LIN {X 0,Y 368.997,Z 325.512,A -85,B 0,C 180,E1 -12767.906,E2 -12767.906} C_VEL
LIN {X 0,Y 369.139,Z 325.499,A -85,B 0,C 180,E1 -12771.892,E2 -12771.892} C_VEL
LIN {X 0,Y 369.12,Z 325.495,A -85,B 0,C 180,E1 -12774.537,E2 -12774.537} C_VEL
LIN {X 0,Y 369.293,Z 325.485,A -85,B 0,C 180,E1 -12777.819,E2 -12777.819} C_VEL
LIN {X 0,Y 369.298,Z 325.479,A -85,B 0,C 180,E1 -12782.181,E2 -12782.181} C_VEL
LIN {X 0,Y 369.147,Z 325.492,A -85,B 0,C 180,E1 -12786.559,E2 -12786.559} C_VEL
LIN {X 0,Y 369.056,Z 325.512,A -85,B 0,C 180,E1 -12789.869,E2 -12789.869} C_VEL
LIN {X 0,Y 369.031,Z 325.503,A -85,B 0,C 180,E1 -12793.772,E2 -12793.772} C_VEL
LIN {X 0,Y 368.985,Z 325.524,A -85,B 0,C 180,E1 -12797.743,E2 -12797.743} C_VEL
LIN {X 0,Y 368.904,Z 325.52,A -85,B 0,C 180,E1 -12801.221,E2 -12801.221} C_VEL
LIN {X 0,Y 368.905,Z 325.533,A -85,B 0,C 180,E1 -12803.875,E2 -12803.875} C_VEL
LIN {X 0,Y 368.852,Z 325.519,A -85,B 0,C 180,E1 -12807.213,E2 -12807.213} C_VEL
LIN {X 0,Y 368.887,Z 325.493,A -85,B 0,C 180,E1 -12809.693,E2 -12809.693} C_VEL
LIN {X 0,Y 368.891,Z 325.526,A -85,B 0,C 180,E1 -12813.043,E2 -12813.043} C_VEL
LIN {X 0,Y 368.911,Z 325.525,A -85,B 0,C 180,E1 -12816.198,E2 -12816.198} C_VEL
LIN {X 0,Y 368.869,Z 325.507,A -85,B 0,C 180,E1 -12818.958,E2 -12818.958} C_VEL
LIN {X 0,Y 368.855,Z 325.537,A -85,B 0,C 180,E1 -12822.006,E2 -12822.006} C_VEL
LIN {X 0,Y 368.87,Z 325.527,A -85,B 0,C 180,E1 -12825.175,E2 -12825.175} C_VEL
LIN {X 0,Y 368.857,Z 325.529,A -85,B 0,C 180,E1 -12828.175,E2 -12828.175} C_VEL
LIN {X 0,Y 368.874,Z 325.529,A -85,B 0,C 180,E1 -12831.367,E2 -12831.367} C_VEL
LIN {X 0,Y 368.929,Z 325.531,A -85,B 0,C 180,E1 -12835.146,E2 -12835.146} C_VEL
LIN {X 0,Y 368.912,Z 325.531,A -85,B 0,C 180,E1 -12839.046,E2 -12839.046} C_VEL
LIN {X 0,Y 368.906,Z 325.505,A -85,B 0,C 180,E1 -12841.558,E2 -12841.558} C_VEL
LIN {X 0,Y 368.922,Z 325.534,A -85,B 0,C 180,E1 -12845.223,E2 -12845.223} C_VEL
LIN {X 0,Y 368.933,Z 325.664,A -85,B 0,C 180,E1 -12848.554,E2 -12848.554} C_VEL
LIN {X 0,Y 369.139,Z 326.592,A -85,B 0,C 180,E1 -12848.752,E2 -12848.752} C_VEL
LIN {X 0,Y 377.458,Z 346.32,A -85,B 0,C 180,E1 -12849.683,E2 -12849.683} C_VEL
LIN {X 0,Y 376.795,Z 405.29,A -85,B 0,C 180,E1 -12850.834,E2 -12850.834} C_VEL
LIN {X 0,Y 376.624,Z 418.447,A -85,B 0,C 180,E1 -12851.267,E2 -12851.267} C_VEL
LIN {X 0,Y 376.25,Z 430.983,A -85,B 0,C 180,E1 -12851.909,E2 -12851.909} C_VEL
LIN {X 0,Y 375.666,Z 442.722,A -85,B 0,C 180,E1 -12852.722,E2 -12852.722} C_VEL
LIN {X 0,Y 374.827,Z 453.399,A -85,B 0,C 180,E1 -12853.666,E2 -12853.666} C_VEL
LIN {X 0,Y 373.891,Z 464.248,A -85,B 0,C 180,E1 -12854.882,E2 -12854.882} C_VEL
LIN {X 0,Y 373.107,Z 473.023,A -85,B 0,C 180,E1 -12856.104,E2 -12856.104} C_VEL
LIN {X 0,Y 372.364,Z 481.054,A -85,B 0,C 180,E1 -12857.464,E2 -12857.464} C_VEL
LIN {X 0,Y 371.492,Z 488.922,A -85,B 0,C 180,E1 -12859.095,E2 -12859.095} C_VEL
LIN {X 0,Y 370.759,Z 494.835,A -85,B 0,C 180,E1 -12860.615,E2 -12860.615} C_VEL
LIN {X 0,Y 370.256,Z 500.214,A -85,B 0,C 180,E1 -12862.365,E2 -12862.365} C_VEL
LIN {X 0,Y 369.648,Z 504.11,A -85,B 0,C 180,E1 -12863.998,E2 -12863.998} C_VEL
LIN {X 0,Y 369.219,Z 506.981,A -85,B 0,C 180,E1 -12865.633,E2 -12865.633} C_VEL
LIN {X 0,Y 369.225,Z 508.328,A -85,B 0,C 180,E1 -12866.727,E2 -12866.727} C_VEL
LIN {X 0,Y 369.048,Z 509.31,A -85,B 0,C 180,E1 -12867.817,E2 -12867.817} C_VEL
LIN {X 0,Y 369.11,Z 509.891,A -85,B 0,C 180,E1 -12868.909,E2 -12868.909} C_VEL
LIN {X 0,Y 369.091,Z 510.119,A -85,B 0,C 180,E1 -12870,E2 -12870} C_VEL
LIN {X 0,Y 369.11,Z 509.934,A -85,B 0,C 180,E1 -12871.091,E2 -12871.091} C_VEL
LIN {X 0,Y 369.047,Z 509.38,A -85,B 0,C 180,E1 -12872.183,E2 -12872.183} C_VEL
LIN {X 0,Y 369.221,Z 508.427,A -85,B 0,C 180,E1 -12873.274,E2 -12873.274} C_VEL
LIN {X 0,Y 369.209,Z 507.125,A -85,B 0,C 180,E1 -12874.367,E2 -12874.367} C_VEL
LIN {X 0,Y 369.643,Z 504.306,A -85,B 0,C 180,E1 -12876.002,E2 -12876.002} C_VEL
LIN {X 0,Y 370.232,Z 500.48,A -85,B 0,C 180,E1 -12877.636,E2 -12877.636} C_VEL
LIN {X 0,Y 370.699,Z 495.402,A -85,B 0,C 180,E1 -12879.328,E2 -12879.328} C_VEL
LIN {X 0,Y 371.612,Z 488.165,A -85,B 0,C 180,E1 -12881.177,E2 -12881.177} C_VEL
LIN {X 0,Y 372.522,Z 480.138,A -85,B 0,C 180,E1 -12882.807,E2 -12882.807} C_VEL
LIN {X 0,Y 373.293,Z 471.916,A -85,B 0,C 180,E1 -12884.167,E2 -12884.167} C_VEL
LIN {X 0,Y 374.07,Z 462.889,A -85,B 0,C 180,E1 -12885.389,E2 -12885.389} C_VEL
LIN {X 0,Y 375.061,Z 452.378,A -85,B 0,C 180,E1 -12886.527,E2 -12886.527} C_VEL
LIN {X 0,Y 375.803,Z 440.712,A -85,B 0,C 180,E1 -12887.537,E2 -12887.537} C_VEL
LIN {X 0,Y 376.419,Z 429.269,A -85,B 0,C 180,E1 -12888.294,E2 -12888.294} C_VEL
LIN {X 0,Y 376.696,Z 416.398,A -85,B 0,C 180,E1 -12888.915,E2 -12888.915} C_VEL
LIN {X 0,Y 376.801,Z 402.594,A -85,B 0,C 180,E1 -12889.333,E2 -12889.333} C_VEL
LIN {X 0,Y 376.774,Z 399.485,A -85,B 0,C 180,E1 -12889.399,E2 -12889.399} C_VEL
LIN {X 0,Y 376.147,Z 393.69,A -85,B 0,C 180,E1 -12889.55,E2 -12889.55} C_VEL
LIN {X 0,Y 371.047,Z 375.043,A -85,B 0,C 180,E1 -12890.224,E2 -12890.224} C_VEL
LIN {X 0,Y 370.502,Z 369.246,A -85,B 0,C 180,E1 -12890.375,E2 -12890.375} C_VEL
LIN {X 0,Y 370.808,Z 347.992,A -85,B 0,C 180,E1 -12890.79,E2 -12890.79} C_VEL
LIN {X 0,Y 362.473,Z 328.467,A -85,B 0,C 180,E1 -12891.729,E2 -12891.729} C_VEL
LIN {X 0,Y 361.96,Z 326.942,A -85,B 0,C 180,E1 -12891.863,E2 -12891.863} C_VEL
LIN {X 0,Y 361.876,Z 326.425,A -85,B 0,C 180,E1 -12892.096,E2 -12892.096} C_VEL
LIN {X 0,Y 361.879,Z 326.4,A -85,B 0,C 180,E1 -12895.293,E2 -12895.293} C_VEL
LIN {X 0,Y 361.855,Z 326.391,A -85,B 0,C 180,E1 -12899.073,E2 -12899.073} C_VEL
LIN {X 0,Y 361.844,Z 326.402,A -85,B 0,C 180,E1 -12902.944,E2 -12902.944} C_VEL
LIN {X 0,Y 361.862,Z 326.408,A -85,B 0,C 180,E1 -12905.637,E2 -12905.637} C_VEL
LIN {X 0,Y 361.823,Z 326.411,A -85,B 0,C 180,E1 -12909.017,E2 -12909.017} C_VEL
LIN {X 0,Y 361.826,Z 326.393,A -85,B 0,C 180,E1 -12912.829,E2 -12912.829} C_VEL
LIN {X 0,Y 361.81,Z 326.414,A -85,B 0,C 180,E1 -12915.947,E2 -12915.947} C_VEL
LIN {X 0,Y 361.806,Z 326.401,A -85,B 0,C 180,E1 -12919.249,E2 -12919.249} C_VEL
LIN {X 0,Y 361.859,Z 326.397,A -85,B 0,C 180,E1 -12922.981,E2 -12922.981} C_VEL
LIN {X 0,Y 361.854,Z 326.406,A -85,B 0,C 180,E1 -12926.63,E2 -12926.63} C_VEL
LIN {X 0,Y 361.842,Z 326.373,A -85,B 0,C 180,E1 -12929.669,E2 -12929.669} C_VEL
LIN {X 0,Y 361.849,Z 326.4,A -85,B 0,C 180,E1 -12933.467,E2 -12933.467} C_VEL
LIN {X 0,Y 361.855,Z 326.406,A -85,B 0,C 180,E1 -12937.142,E2 -12937.142} C_VEL
LIN {X 0,Y 361.869,Z 326.407,A -85,B 0,C 180,E1 -12940.721,E2 -12940.721} C_VEL
LIN {X 0,Y 361.933,Z 326.393,A -85,B 0,C 180,E1 -12944.225,E2 -12944.225} C_VEL
LIN {X 0,Y 361.993,Z 326.384,A -85,B 0,C 180,E1 -12946.527,E2 -12946.527} C_VEL
LIN {X 0,Y 361.99,Z 326.392,A -85,B 0,C 180,E1 -12949.937,E2 -12949.937} C_VEL
LIN {X 0,Y 362.108,Z 326.37,A -85,B 0,C 180,E1 -12953.313,E2 -12953.313} C_VEL
LIN {X 0,Y 362.261,Z 326.355,A -85,B 0,C 180,E1 -12957.776,E2 -12957.776} C_VEL
LIN {X 0,Y 362.256,Z 326.361,A -85,B 0,C 180,E1 -12962.224,E2 -12962.224} C_VEL
LIN {X 0,Y 362.133,Z 326.364,A -85,B 0,C 180,E1 -12966.687,E2 -12966.687} C_VEL
LIN {X 0,Y 361.989,Z 326.395,A -85,B 0,C 180,E1 -12970.063,E2 -12970.063} C_VEL
LIN {X 0,Y 361.992,Z 326.382,A -85,B 0,C 180,E1 -12973.899,E2 -12973.899} C_VEL
LIN {X 0,Y 361.922,Z 326.399,A -85,B 0,C 180,E1 -12976.935,E2 -12976.935} C_VEL
LIN {X 0,Y 361.877,Z 326.381,A -85,B 0,C 180,E1 -12980.461,E2 -12980.461} C_VEL
LIN {X 0,Y 361.855,Z 326.41,A -85,B 0,C 180,E1 -12984.102,E2 -12984.102} C_VEL
LIN {X 0,Y 361.837,Z 326.397,A -85,B 0,C 180,E1 -12987.785,E2 -12987.785} C_VEL
LIN {X 0,Y 361.842,Z 326.411,A -85,B 0,C 180,E1 -12991.286,E2 -12991.286} C_VEL
LIN {X 0,Y 361.846,Z 326.399,A -85,B 0,C 180,E1 -12994.281,E2 -12994.281} C_VEL
LIN {X 0,Y 361.852,Z 326.41,A -85,B 0,C 180,E1 -12997.222,E2 -12997.222} C_VEL
LIN {X 0,Y 361.807,Z 326.416,A -85,B 0,C 180,E1 -13000.751,E2 -13000.751} C_VEL
LIN {X 0,Y 361.806,Z 326.386,A -85,B 0,C 180,E1 -13004.37,E2 -13004.37} C_VEL
LIN {X 0,Y 361.819,Z 326.414,A -85,B 0,C 180,E1 -13007.571,E2 -13007.571} C_VEL
LIN {X 0,Y 361.839,Z 326.402,A -85,B 0,C 180,E1 -13011.572,E2 -13011.572} C_VEL
LIN {X 0,Y 361.91,Z 326.58,A -85,B 0,C 180,E1 -13014.953,E2 -13014.953} C_VEL
LIN {X 0,Y 364.912,Z 338.861,A -85,B 0,C 180,E1 -13017.597,E2 -13017.597} C_VEL
LIN {X 0,Y 367.691,Z 351.772,A -85,B 0,C 180,E1 -13020.201,E2 -13020.201} C_VEL
LIN {X 0,Y 367.318,Z 358.573,A -85,B 0,C 180,E1 -13021.424,E2 -13021.424} C_VEL
LIN {X 0,Y 365.124,Z 381.961,A -85,B 0,C 180,E1 -13025.554,E2 -13025.554} C_VEL
LIN {X 0,Y 364.057,Z 395.066,A -85,B 0,C 180,E1 -13027.831,E2 -13027.831} C_VEL
LIN {X 0,Y 367.984,Z 428.586,A -85,B 0,C 180,E1 -13028.774,E2 -13028.774} C_VEL
LIN {X 0,Y 369.463,Z 445.477,A -85,B 0,C 180,E1 -13029.201,E2 -13029.201} C_VEL
LIN {X 0,Y 368.499,Z 505.753,A -85,B 0,C 180,E1 -13030.395,E2 -13030.395} C_VEL
LIN {X 0,Y 367.813,Z 519.02,A -85,B 0,C 180,E1 -13030.864,E2 -13030.864} C_VEL
LIN {X 0,Y 366.828,Z 532.347,A -85,B 0,C 180,E1 -13031.572,E2 -13031.572} C_VEL
LIN {X 0,Y 365.679,Z 543.548,A -85,B 0,C 180,E1 -13032.38,E2 -13032.38} C_VEL
LIN {X 0,Y 364.475,Z 555.248,A -85,B 0,C 180,E1 -13033.476,E2 -13033.476} C_VEL
LIN {X 0,Y 363.415,Z 564.724,A -85,B 0,C 180,E1 -13034.579,E2 -13034.579} C_VEL
LIN {X 0,Y 362.436,Z 574.494,A -85,B 0,C 180,E1 -13035.973,E2 -13035.973} C_VEL
LIN {X 0,Y 361.919,Z 581.022,A -85,B 0,C 180,E1 -13037.096,E2 -13037.096} C_VEL
LIN {X 0,Y 361.274,Z 589.239,A -85,B 0,C 180,E1 -13038.783,E2 -13038.783} C_VEL
LIN {X 0,Y 360.931,Z 595.87,A -85,B 0,C 180,E1 -13040.473,E2 -13040.473} C_VEL
LIN {X 0,Y 360.895,Z 601.177,A -85,B 0,C 180,E1 -13042.165,E2 -13042.165} C_VEL
LIN {X 0,Y 361.013,Z 605.321,A -85,B 0,C 180,E1 -13043.854,E2 -13043.854} C_VEL
LIN {X 0,Y 361.197,Z 608.397,A -85,B 0,C 180,E1 -13045.536,E2 -13045.536} C_VEL
LIN {X 0,Y 361.295,Z 609.864,A -85,B 0,C 180,E1 -13046.655,E2 -13046.655} C_VEL
LIN {X 0,Y 361.693,Z 611.588,A -85,B 0,C 180,E1 -13048.887,E2 -13048.887} C_VEL
LIN {X 0,Y 361.754,Z 611.819,A -85,B 0,C 180,E1 -13050,E2 -13050} C_VEL
LIN {X 0,Y 361.694,Z 611.584,A -85,B 0,C 180,E1 -13051.113,E2 -13051.113} C_VEL
LIN {X 0,Y 361.299,Z 609.858,A -85,B 0,C 180,E1 -13053.345,E2 -13053.345} C_VEL
LIN {X 0,Y 361.21,Z 608.388,A -85,B 0,C 180,E1 -13054.464,E2 -13054.464} C_VEL
LIN {X 0,Y 361.035,Z 605.305,A -85,B 0,C 180,E1 -13056.146,E2 -13056.146} C_VEL
LIN {X 0,Y 360.904,Z 601.15,A -85,B 0,C 180,E1 -13057.834,E2 -13057.834} C_VEL
LIN {X 0,Y 360.973,Z 594.801,A -85,B 0,C 180,E1 -13059.808,E2 -13059.808} C_VEL
LIN {X 0,Y 361.376,Z 587.926,A -85,B 0,C 180,E1 -13061.498,E2 -13061.498} C_VEL
LIN {X 0,Y 361.914,Z 580.962,A -85,B 0,C 180,E1 -13062.904,E2 -13062.904} C_VEL
LIN {X 0,Y 362.7,Z 571.813,A -85,B 0,C 180,E1 -13064.427,E2 -13064.427} C_VEL
LIN {X 0,Y 363.585,Z 562.451,A -85,B 0,C 180,E1 -13065.701,E2 -13065.701} C_VEL
LIN {X 0,Y 364.898,Z 551.055,A -85,B 0,C 180,E1 -13066.936,E2 -13066.936} C_VEL
LIN {X 0,Y 366.036,Z 539.916,A -85,B 0,C 180,E1 -13067.891,E2 -13067.891} C_VEL
LIN {X 0,Y 367.224,Z 527.607,A -85,B 0,C 180,E1 -13068.697,E2 -13068.697} C_VEL
LIN {X 0,Y 368.076,Z 514.653,A -85,B 0,C 180,E1 -13069.303,E2 -13069.303} C_VEL
LIN {X 0,Y 368.541,Z 500.894,A -85,B 0,C 180,E1 -13069.712,E2 -13069.712} C_VEL
LIN {X 0,Y 369.37,Z 443.517,A -85,B 0,C 180,E1 -13070.83,E2 -13070.83} C_VEL
LIN {X 0,Y 365.882,Z 410.175,A -85,B 0,C 180,E1 -13071.711,E2 -13071.711} C_VEL
LIN {X 0,Y 364.018,Z 394.864,A -85,B 0,C 180,E1 -13072.173,E2 -13072.173} C_VEL
LIN {X 0,Y 365.701,Z 374.774,A -85,B 0,C 180,E1 -13075.703,E2 -13075.703} C_VEL
LIN {X 0,Y 367.61,Z 355.111,A -85,B 0,C 180,E1 -13079.176,E2 -13079.176} C_VEL
LIN {X 0,Y 367.643,Z 351.679,A -85,B 0,C 180,E1 -13079.803,E2 -13079.803} C_VEL
LIN {X 0,Y 364.613,Z 337.52,A -85,B 0,C 180,E1 -13082.663,E2 -13082.663} C_VEL
LIN {X 0,Y 361.91,Z 326.536,A -85,B 0,C 180,E1 -13085.047,E2 -13085.047} C_VEL
LIN {X 0,Y 361.839,Z 326.403,A -85,B 0,C 180,E1 -13088.428,E2 -13088.428} C_VEL
LIN {X 0,Y 361.819,Z 326.415,A -85,B 0,C 180,E1 -13092.429,E2 -13092.429} C_VEL
LIN {X 0,Y 361.808,Z 326.39,A -85,B 0,C 180,E1 -13095.947,E2 -13095.947} C_VEL
LIN {X 0,Y 361.807,Z 326.417,A -85,B 0,C 180,E1 -13099.249,E2 -13099.249} C_VEL
LIN {X 0,Y 361.855,Z 326.355,A -85,B 0,C 180,E1 -13102.98,E2 -13102.98} C_VEL
LIN {X 0,Y 361.853,Z 326.406,A -85,B 0,C 180,E1 -13106.631,E2 -13106.631} C_VEL
LIN {X 0,Y 361.851,Z 326.406,A -85,B 0,C 180,E1 -13109.67,E2 -13109.67} C_VEL
LIN {X 0,Y 361.86,Z 326.403,A -85,B 0,C 180,E1 -13113.468,E2 -13113.468} C_VEL
LIN {X 0,Y 361.87,Z 326.403,A -85,B 0,C 180,E1 -13117.143,E2 -13117.143} C_VEL
LIN {X 0,Y 361.898,Z 326.39,A -85,B 0,C 180,E1 -13120.723,E2 -13120.723} C_VEL
LIN {X 0,Y 361.927,Z 326.399,A -85,B 0,C 180,E1 -13123.066,E2 -13123.066} C_VEL
LIN {X 0,Y 361.993,Z 326.379,A -85,B 0,C 180,E1 -13126.528,E2 -13126.528} C_VEL
LIN {X 0,Y 361.992,Z 326.396,A -85,B 0,C 180,E1 -13129.937,E2 -13129.937} C_VEL
LIN {X 0,Y 362.134,Z 326.365,A -85,B 0,C 180,E1 -13133.313,E2 -13133.313} C_VEL
LIN {X 0,Y 362.256,Z 326.362,A -85,B 0,C 180,E1 -13137.776,E2 -13137.776} C_VEL
LIN {X 0,Y 362.261,Z 326.355,A -85,B 0,C 180,E1 -13142.224,E2 -13142.224} C_VEL
LIN {X 0,Y 362.111,Z 326.369,A -85,B 0,C 180,E1 -13146.687,E2 -13146.687} C_VEL
LIN {X 0,Y 361.993,Z 326.392,A -85,B 0,C 180,E1 -13150.063,E2 -13150.063} C_VEL
LIN {X 0,Y 361.992,Z 326.379,A -85,B 0,C 180,E1 -13153.899,E2 -13153.899} C_VEL
LIN {X 0,Y 361.921,Z 326.398,A -85,B 0,C 180,E1 -13156.935,E2 -13156.935} C_VEL
LIN {X 0,Y 361.877,Z 326.395,A -85,B 0,C 180,E1 -13160.462,E2 -13160.462} C_VEL
LIN {X 0,Y 361.856,Z 326.409,A -85,B 0,C 180,E1 -13164.102,E2 -13164.102} C_VEL
LIN {X 0,Y 361.829,Z 326.385,A -85,B 0,C 180,E1 -13167.786,E2 -13167.786} C_VEL
LIN {X 0,Y 361.84,Z 326.383,A -85,B 0,C 180,E1 -13171.285,E2 -13171.285} C_VEL
LIN {X 0,Y 361.849,Z 326.41,A -85,B 0,C 180,E1 -13174.281,E2 -13174.281} C_VEL
LIN {X 0,Y 361.855,Z 326.396,A -85,B 0,C 180,E1 -13177.222,E2 -13177.222} C_VEL
LIN {X 0,Y 361.806,Z 326.399,A -85,B 0,C 180,E1 -13180.751,E2 -13180.751} C_VEL
LIN {X 0,Y 361.809,Z 326.413,A -85,B 0,C 180,E1 -13184.37,E2 -13184.37} C_VEL
LIN {X 0,Y 361.819,Z 326.396,A -85,B 0,C 180,E1 -13187.571,E2 -13187.571} C_VEL
LIN {X 0,Y 361.84,Z 326.402,A -85,B 0,C 180,E1 -13191.573,E2 -13191.573} C_VEL
LIN {X 0,Y 361.868,Z 326.407,A -85,B 0,C 180,E1 -13194.657,E2 -13194.657} C_VEL
LIN {X 0,Y 361.836,Z 326.409,A -85,B 0,C 180,E1 -13198.371,E2 -13198.371} C_VEL
LIN {X 0,Y 361.848,Z 326.394,A -85,B 0,C 180,E1 -13200.951,E2 -13200.951} C_VEL
LIN {X 0,Y 361.879,Z 326.4,A -85,B 0,C 180,E1 -13204.707,E2 -13204.707} C_VEL
LIN {X 0,Y 361.903,Z 326.554,A -85,B 0,C 180,E1 -13208.124,E2 -13208.124} C_VEL
LIN {X 0,Y 362.125,Z 327.56,A -85,B 0,C 180,E1 -13208.321,E2 -13208.321} C_VEL
LIN {X 0,Y 369.789,Z 345.481,A -85,B 0,C 180,E1 -13209.201,E2 -13209.201} C_VEL
LIN {X 0,Y 370.86,Z 348.15,A -85,B 0,C 180,E1 -13209.322,E2 -13209.322} C_VEL
LIN {X 0,Y 370.152,Z 405.371,A -85,B 0,C 180,E1 -13210.454,E2 -13210.454} C_VEL
LIN {X 0,Y 369.988,Z 418.734,A -85,B 0,C 180,E1 -13210.889,E2 -13210.889} C_VEL
LIN {X 0,Y 369.616,Z 430.853,A -85,B 0,C 180,E1 -13211.501,E2 -13211.501} C_VEL
LIN {X 0,Y 368.981,Z 443.151,A -85,B 0,C 180,E1 -13212.354,E2 -13212.354} C_VEL
LIN {X 0,Y 368.203,Z 453.321,A -85,B 0,C 180,E1 -13213.256,E2 -13213.256} C_VEL
LIN {X 0,Y 367.184,Z 464.17,A -85,B 0,C 180,E1 -13214.457,E2 -13214.457} C_VEL
LIN {X 0,Y 366.288,Z 474.004,A -85,B 0,C 180,E1 -13215.84,E2 -13215.84} C_VEL
LIN {X 0,Y 365.506,Z 482.035,A -85,B 0,C 180,E1 -13217.225,E2 -13217.225} C_VEL
LIN {X 0,Y 364.594,Z 489.902,A -85,B 0,C 180,E1 -13218.886,E2 -13218.886} C_VEL
LIN {X 0,Y 363.827,Z 495.815,A -85,B 0,C 180,E1 -13220.435,E2 -13220.435} C_VEL
LIN {X 0,Y 363.292,Z 501.193,A -85,B 0,C 180,E1 -13222.217,E2 -13222.217} C_VEL
LIN {X 0,Y 362.659,Z 505.088,A -85,B 0,C 180,E1 -13223.882,E2 -13223.882} C_VEL
LIN {X 0,Y 362.208,Z 507.96,A -85,B 0,C 180,E1 -13225.549,E2 -13225.549} C_VEL
LIN {X 0,Y 362.207,Z 509.307,A -85,B 0,C 180,E1 -13226.663,E2 -13226.663} C_VEL
LIN {X 0,Y 362.026,Z 510.288,A -85,B 0,C 180,E1 -13227.775,E2 -13227.775} C_VEL
LIN {X 0,Y 362.085,Z 510.869,A -85,B 0,C 180,E1 -13228.888,E2 -13228.888} C_VEL
LIN {X 0,Y 362.065,Z 511.097,A -85,B 0,C 180,E1 -13230,E2 -13230} C_VEL
LIN {X 0,Y 362.085,Z 510.911,A -85,B 0,C 180,E1 -13231.112,E2 -13231.112} C_VEL
LIN {X 0,Y 362.025,Z 510.358,A -85,B 0,C 180,E1 -13232.225,E2 -13232.225} C_VEL
LIN {X 0,Y 362.204,Z 509.404,A -85,B 0,C 180,E1 -13233.337,E2 -13233.337} C_VEL
LIN {X 0,Y 362.198,Z 508.103,A -85,B 0,C 180,E1 -13234.451,E2 -13234.451} C_VEL
LIN {X 0,Y 362.654,Z 505.283,A -85,B 0,C 180,E1 -13236.118,E2 -13236.118} C_VEL
LIN {X 0,Y 363.268,Z 501.457,A -85,B 0,C 180,E1 -13237.783,E2 -13237.783} C_VEL
LIN {X 0,Y 363.765,Z 496.379,A -85,B 0,C 180,E1 -13239.508,E2 -13239.508} C_VEL
LIN {X 0,Y 364.723,Z 489.141,A -85,B 0,C 180,E1 -13241.391,E2 -13241.391} C_VEL
LIN {X 0,Y 365.671,Z 481.113,A -85,B 0,C 180,E1 -13243.051,E2 -13243.051} C_VEL
LIN {X 0,Y 366.481,Z 472.892,A -85,B 0,C 180,E1 -13244.436,E2 -13244.436} C_VEL
LIN {X 0,Y 367.311,Z 463.861,A -85,B 0,C 180,E1 -13245.68,E2 -13245.68} C_VEL
LIN {X 0,Y 368.325,Z 453.353,A -85,B 0,C 180,E1 -13246.838,E2 -13246.838} C_VEL
LIN {X 0,Y 369.087,Z 441.84,A -85,B 0,C 180,E1 -13247.854,E2 -13247.854} C_VEL
LIN {X 0,Y 369.732,Z 430.576,A -85,B 0,C 180,E1 -13248.616,E2 -13248.616} C_VEL
LIN {X 0,Y 370.095,Z 418.263,A -85,B 0,C 180,E1 -13249.229,E2 -13249.229} C_VEL
LIN {X 0,Y 370.183,Z 408.012,A -85,B 0,C 180,E1 -13249.585,E2 -13249.585} C_VEL
LIN {X 0,Y 370.502,Z 369.246,A -85,B 0,C 180,E1 -13250.375,E2 -13250.375} C_VEL
LIN {X 0,Y 370.017,Z 365.384,A -85,B 0,C 180,E1 -13250.483,E2 -13250.483} C_VEL
LIN {X 0,Y 367.762,Z 359.348,A -85,B 0,C 180,E1 -13250.745,E2 -13250.745} C_VEL
LIN {X 0,Y 364.755,Z 352.129,A -85,B 0,C 180,E1 -13251.083,E2 -13251.083} C_VEL
LIN {X 0,Y 364.157,Z 349.57,A -85,B 0,C 180,E1 -13251.175,E2 -13251.175} C_VEL
LIN {X 0,Y 355.034,Z 328.299,A -85,B 0,C 180,E1 -13252.254,E2 -13252.254} C_VEL
LIN {X 0,Y 354.823,Z 327.338,A -85,B 0,C 180,E1 -13252.487,E2 -13252.487} C_VEL
LIN {X 0,Y 354.808,Z 327.266,A -85,B 0,C 180,E1 -13255.834,E2 -13255.834} C_VEL
LIN {X 0,Y 354.792,Z 327.283,A -85,B 0,C 180,E1 -13259.684,E2 -13259.684} C_VEL
LIN {X 0,Y 354.783,Z 327.281,A -85,B 0,C 180,E1 -13262.333,E2 -13262.333} C_VEL
LIN {X 0,Y 354.817,Z 327.285,A -85,B 0,C 180,E1 -13265.698,E2 -13265.698} C_VEL
LIN {X 0,Y 354.766,Z 327.293,A -85,B 0,C 180,E1 -13269.412,E2 -13269.412} C_VEL
LIN {X 0,Y 354.778,Z 327.27,A -85,B 0,C 180,E1 -13272.865,E2 -13272.865} C_VEL
LIN {X 0,Y 354.759,Z 327.293,A -85,B 0,C 180,E1 -13276.102,E2 -13276.102} C_VEL
LIN {X 0,Y 354.759,Z 327.279,A -85,B 0,C 180,E1 -13279.175,E2 -13279.175} C_VEL
LIN {X 0,Y 354.796,Z 327.268,A -85,B 0,C 180,E1 -13282.404,E2 -13282.404} C_VEL
LIN {X 0,Y 354.807,Z 327.289,A -85,B 0,C 180,E1 -13284.94,E2 -13284.94} C_VEL
LIN {X 0,Y 354.785,Z 327.266,A -85,B 0,C 180,E1 -13288.406,E2 -13288.406} C_VEL
LIN {X 0,Y 354.783,Z 327.256,A -85,B 0,C 180,E1 -13291.613,E2 -13291.613} C_VEL
LIN {X 0,Y 354.798,Z 327.287,A -85,B 0,C 180,E1 -13295.419,E2 -13295.419} C_VEL
LIN {X 0,Y 354.816,Z 327.275,A -85,B 0,C 180,E1 -13299.112,E2 -13299.112} C_VEL
LIN {X 0,Y 354.872,Z 327.279,A -85,B 0,C 180,E1 -13302.718,E2 -13302.718} C_VEL
LIN {X 0,Y 354.945,Z 327.258,A -85,B 0,C 180,E1 -13306.255,E2 -13306.255} C_VEL
LIN {X 0,Y 354.947,Z 327.269,A -85,B 0,C 180,E1 -13309.735,E2 -13309.735} C_VEL
LIN {X 0,Y 355.075,Z 327.246,A -85,B 0,C 180,E1 -13313.179,E2 -13313.179} C_VEL
LIN {X 0,Y 355.223,Z 327.231,A -85,B 0,C 180,E1 -13317.732,E2 -13317.732} C_VEL
LIN {X 0,Y 355.218,Z 327.238,A -85,B 0,C 180,E1 -13322.268,E2 -13322.268} C_VEL
LIN {X 0,Y 355.096,Z 327.241,A -85,B 0,C 180,E1 -13326.82,E2 -13326.82} C_VEL
LIN {X 0,Y 354.945,Z 327.271,A -85,B 0,C 180,E1 -13330.265,E2 -13330.265} C_VEL
LIN {X 0,Y 354.937,Z 327.262,A -85,B 0,C 180,E1 -13334.019,E2 -13334.019} C_VEL
LIN {X 0,Y 354.884,Z 327.271,A -85,B 0,C 180,E1 -13338.092,E2 -13338.092} C_VEL
LIN {X 0,Y 354.813,Z 327.264,A -85,B 0,C 180,E1 -13341.418,E2 -13341.418} C_VEL
LIN {X 0,Y 354.8,Z 327.29,A -85,B 0,C 180,E1 -13344.581,E2 -13344.581} C_VEL
LIN {X 0,Y 354.795,Z 327.271,A -85,B 0,C 180,E1 -13348.386,E2 -13348.386} C_VEL
LIN {X 0,Y 354.782,Z 327.291,A -85,B 0,C 180,E1 -13352.334,E2 -13352.334} C_VEL
LIN {X 0,Y 354.813,Z 327.279,A -85,B 0,C 180,E1 -13355.699,E2 -13355.699} C_VEL
LIN {X 0,Y 354.764,Z 327.283,A -85,B 0,C 180,E1 -13359.413,E2 -13359.413} C_VEL
LIN {X 0,Y 354.779,Z 327.285,A -85,B 0,C 180,E1 -13362.867,E2 -13362.867} C_VEL
LIN {X 0,Y 354.758,Z 327.269,A -85,B 0,C 180,E1 -13366.103,E2 -13366.103} C_VEL
LIN {X 0,Y 354.76,Z 327.284,A -85,B 0,C 180,E1 -13369.176,E2 -13369.176} C_VEL
LIN {X 0,Y 354.796,Z 327.293,A -85,B 0,C 180,E1 -13372.405,E2 -13372.405} C_VEL
LIN {X 0,Y 354.869,Z 327.474,A -85,B 0,C 180,E1 -13374.54,E2 -13374.54} C_VEL
LIN {X 0,Y 358.194,Z 341.109,A -85,B 0,C 180,E1 -13377.532,E2 -13377.532} C_VEL
LIN {X 0,Y 360.646,Z 352.499,A -85,B 0,C 180,E1 -13379.882,E2 -13379.882} C_VEL
LIN {X 0,Y 360.778,Z 355.937,A -85,B 0,C 180,E1 -13380.537,E2 -13380.537} C_VEL
LIN {X 0,Y 359.046,Z 372.677,A -85,B 0,C 180,E1 -13383.558,E2 -13383.558} C_VEL
LIN {X 0,Y 357.397,Z 390.803,A -85,B 0,C 180,E1 -13386.841,E2 -13386.841} C_VEL
LIN {X 0,Y 357.19,Z 393.844,A -85,B 0,C 180,E1 -13387.365,E2 -13387.365} C_VEL
LIN {X 0,Y 361.291,Z 428.682,A -85,B 0,C 180,E1 -13388.384,E2 -13388.384} C_VEL
LIN {X 0,Y 362.795,Z 446.41,A -85,B 0,C 180,E1 -13388.84,E2 -13388.84} C_VEL
LIN {X 0,Y 361.789,Z 504.774,A -85,B 0,C 180,E1 -13390.016,E2 -13390.016} C_VEL
LIN {X 0,Y 361.085,Z 518.037,A -85,B 0,C 180,E1 -13390.493,E2 -13390.493} C_VEL
LIN {X 0,Y 360.058,Z 531.359,A -85,B 0,C 180,E1 -13391.212,E2 -13391.212} C_VEL
LIN {X 0,Y 358.911,Z 542.563,A -85,B 0,C 180,E1 -13392.037,E2 -13392.037} C_VEL
LIN {X 0,Y 357.681,Z 554.265,A -85,B 0,C 180,E1 -13393.153,E2 -13393.153} C_VEL
LIN {X 0,Y 356.409,Z 564.819,A -85,B 0,C 180,E1 -13394.415,E2 -13394.415} C_VEL
LIN {X 0,Y 355.376,Z 574.495,A -85,B 0,C 180,E1 -13395.855,E2 -13395.855} C_VEL
LIN {X 0,Y 354.982,Z 580.033,A -85,B 0,C 180,E1 -13396.84,E2 -13396.84} C_VEL
LIN {X 0,Y 354.264,Z 588.246,A -85,B 0,C 180,E1 -13398.558,E2 -13398.558} C_VEL
LIN {X 0,Y 353.886,Z 594.877,A -85,B 0,C 180,E1 -13400.282,E2 -13400.282} C_VEL
LIN {X 0,Y 353.804,Z 600.181,A -85,B 0,C 180,E1 -13402.007,E2 -13402.007} C_VEL
LIN {X 0,Y 353.918,Z 603.896,A -85,B 0,C 180,E1 -13403.529,E2 -13403.529} C_VEL
LIN {X 0,Y 354.132,Z 607.411,A -85,B 0,C 180,E1 -13405.447,E2 -13405.447} C_VEL
LIN {X 0,Y 354.243,Z 608.882,A -85,B 0,C 180,E1 -13406.588,E2 -13406.588} C_VEL
LIN {X 0,Y 354.659,Z 610.609,A -85,B 0,C 180,E1 -13408.865,E2 -13408.865} C_VEL
LIN {X 0,Y 354.728,Z 610.842,A -85,B 0,C 180,E1 -13410,E2 -13410} C_VEL
LIN {X 0,Y 354.659,Z 610.605,A -85,B 0,C 180,E1 -13411.135,E2 -13411.135} C_VEL
LIN {X 0,Y 354.248,Z 608.874,A -85,B 0,C 180,E1 -13413.412,E2 -13413.412} C_VEL
LIN {X 0,Y 354.144,Z 607.401,A -85,B 0,C 180,E1 -13414.553,E2 -13414.553} C_VEL
LIN {X 0,Y 353.926,Z 603.85,A -85,B 0,C 180,E1 -13416.481,E2 -13416.481} C_VEL
LIN {X 0,Y 353.803,Z 598.49,A -85,B 0,C 180,E1 -13418.568,E2 -13418.568} C_VEL
LIN {X 0,Y 353.971,Z 592.76,A -85,B 0,C 180,E1 -13420.293,E2 -13420.293} C_VEL
LIN {X 0,Y 354.416,Z 585.653,A -85,B 0,C 180,E1 -13422.017,E2 -13422.017} C_VEL
LIN {X 0,Y 355.248,Z 576.816,A -85,B 0,C 180,E1 -13423.733,E2 -13423.733} C_VEL
LIN {X 0,Y 356.133,Z 567.789,A -85,B 0,C 180,E1 -13425.157,E2 -13425.157} C_VEL
LIN {X 0,Y 356.964,Z 559.102,A -85,B 0,C 180,E1 -13426.293,E2 -13426.293} C_VEL
LIN {X 0,Y 358.414,Z 547.178,A -85,B 0,C 180,E1 -13427.546,E2 -13427.546} C_VEL
LIN {X 0,Y 359.673,Z 535.194,A -85,B 0,C 180,E1 -13428.513,E2 -13428.513} C_VEL
LIN {X 0,Y 360.745,Z 522.751,A -85,B 0,C 180,E1 -13429.267,E2 -13429.267} C_VEL
LIN {X 0,Y 361.572,Z 509.975,A -85,B 0,C 180,E1 -13429.812,E2 -13429.812} C_VEL
LIN {X 0,Y 361.943,Z 496.531,A -85,B 0,C 180,E1 -13430.161,E2 -13430.161} C_VEL
LIN {X 0,Y 362.709,Z 444.243,A -85,B 0,C 180,E1 -13431.195,E2 -13431.195} C_VEL
LIN {X 0,Y 358.966,Z 408.327,A -85,B 0,C 180,E1 -13432.168,E2 -13432.168} C_VEL
LIN {X 0,Y 357.167,Z 393.83,A -85,B 0,C 180,E1 -13432.624,E2 -13432.624} C_VEL
LIN {X 0,Y 358.86,Z 374.246,A -85,B 0,C 180,E1 -13436.144,E2 -13436.144} C_VEL
LIN {X 0,Y 360.788,Z 355.847,A -85,B 0,C 180,E1 -13439.462,E2 -13439.462} C_VEL
LIN {X 0,Y 360.605,Z 352.396,A -85,B 0,C 180,E1 -13440.122,E2 -13440.122} C_VEL
LIN {X 0,Y 357.792,Z 339.337,A -85,B 0,C 180,E1 -13442.823,E2 -13442.823} C_VEL
LIN {X 0,Y 354.837,Z 327.393,A -85,B 0,C 180,E1 -13445.486,E2 -13445.486} C_VEL
LIN {X 0,Y 354.782,Z 327.273,A -85,B 0,C 180,E1 -13449.337,E2 -13449.337} C_VEL
LIN {X 0,Y 354.778,Z 327.289,A -85,B 0,C 180,E1 -13452.865,E2 -13452.865} C_VEL
LIN {X 0,Y 354.758,Z 327.27,A -85,B 0,C 180,E1 -13456.102,E2 -13456.102} C_VEL
LIN {X 0,Y 354.76,Z 327.294,A -85,B 0,C 180,E1 -13459.175,E2 -13459.175} C_VEL
LIN {X 0,Y 354.794,Z 327.236,A -85,B 0,C 180,E1 -13462.404,E2 -13462.404} C_VEL
LIN {X 0,Y 354.803,Z 327.259,A -85,B 0,C 180,E1 -13464.94,E2 -13464.94} C_VEL
LIN {X 0,Y 354.788,Z 327.29,A -85,B 0,C 180,E1 -13468.405,E2 -13468.405} C_VEL
LIN {X 0,Y 354.796,Z 327.271,A -85,B 0,C 180,E1 -13471.614,E2 -13471.614} C_VEL
LIN {X 0,Y 354.8,Z 327.29,A -85,B 0,C 180,E1 -13475.419,E2 -13475.419} C_VEL
LIN {X 0,Y 354.819,Z 327.259,A -85,B 0,C 180,E1 -13479.113,E2 -13479.113} C_VEL
LIN {X 0,Y 354.893,Z 327.274,A -85,B 0,C 180,E1 -13482.72,E2 -13482.72} C_VEL
LIN {X 0,Y 354.945,Z 327.258,A -85,B 0,C 180,E1 -13486.255,E2 -13486.255} C_VEL
LIN {X 0,Y 354.948,Z 327.271,A -85,B 0,C 180,E1 -13489.735,E2 -13489.735} C_VEL
LIN {X 0,Y 355.098,Z 327.241,A -85,B 0,C 180,E1 -13493.18,E2 -13493.18} C_VEL
LIN {X 0,Y 355.219,Z 327.239,A -85,B 0,C 180,E1 -13497.732,E2 -13497.732} C_VEL
LIN {X 0,Y 355.138,Z 327.23,A -85,B 0,C 180,E1 -13501.134,E2 -13501.134} C_VEL
LIN {X 0,Y 355.224,Z 327.231,A -85,B 0,C 180,E1 -13502.268,E2 -13502.268} C_VEL
LIN {X 0,Y 355.078,Z 327.245,A -85,B 0,C 180,E1 -13506.82,E2 -13506.82} C_VEL
LIN {X 0,Y 354.949,Z 327.268,A -85,B 0,C 180,E1 -13510.265,E2 -13510.265} C_VEL
LIN {X 0,Y 354.937,Z 327.256,A -85,B 0,C 180,E1 -13514.019,E2 -13514.019} C_VEL
LIN {X 0,Y 354.884,Z 327.277,A -85,B 0,C 180,E1 -13518.092,E2 -13518.092} C_VEL
LIN {X 0,Y 354.811,Z 327.276,A -85,B 0,C 180,E1 -13521.417,E2 -13521.417} C_VEL
LIN {X 0,Y 354.798,Z 327.287,A -85,B 0,C 180,E1 -13524.581,E2 -13524.581} C_VEL
LIN {X 0,Y 354.783,Z 327.256,A -85,B 0,C 180,E1 -13528.387,E2 -13528.387} C_VEL
LIN {X 0,Y 354.78,Z 327.28,A -85,B 0,C 180,E1 -13532.334,E2 -13532.334} C_VEL
LIN {X 0,Y 354.817,Z 327.285,A -85,B 0,C 180,E1 -13535.7,E2 -13535.7} C_VEL
LIN {X 0,Y 354.764,Z 327.262,A -85,B 0,C 180,E1 -13539.413,E2 -13539.413} C_VEL
LIN {X 0,Y 354.778,Z 327.291,A -85,B 0,C 180,E1 -13542.867,E2 -13542.867} C_VEL
LIN {X 0,Y 354.759,Z 327.274,A -85,B 0,C 180,E1 -13546.103,E2 -13546.103} C_VEL
LIN {X 0,Y 354.76,Z 327.291,A -85,B 0,C 180,E1 -13549.176,E2 -13549.176} C_VEL
LIN {X 0,Y 354.797,Z 327.273,A -85,B 0,C 180,E1 -13552.405,E2 -13552.405} C_VEL
LIN {X 0,Y 354.807,Z 327.288,A -85,B 0,C 180,E1 -13554.941,E2 -13554.941} C_VEL
LIN {X 0,Y 354.792,Z 327.286,A -85,B 0,C 180,E1 -13558.406,E2 -13558.406} C_VEL
LIN {X 0,Y 354.788,Z 327.261,A -85,B 0,C 180,E1 -13561.614,E2 -13561.614} C_VEL
LIN {X 0,Y 354.835,Z 327.289,A -85,B 0,C 180,E1 -13565.658,E2 -13565.658} C_VEL
LIN {X 0,Y 354.841,Z 327.44,A -85,B 0,C 180,E1 -13567.665,E2 -13567.665} C_VEL
LIN {X 0,Y 355.025,Z 328.338,A -85,B 0,C 180,E1 -13567.854,E2 -13567.854} C_VEL
LIN {X 0,Y 363.198,Z 347.162,A -85,B 0,C 180,E1 -13568.82,E2 -13568.82} C_VEL
LIN {X 0,Y 364.245,Z 349.775,A -85,B 0,C 180,E1 -13568.942,E2 -13568.942} C_VEL
LIN {X 0,Y 363.526,Z 405.452,A -85,B 0,C 180,E1 -13570.06,E2 -13570.06} C_VEL
LIN {X 0,Y 363.409,Z 418.142,A -85,B 0,C 180,E1 -13570.465,E2 -13570.465} C_VEL
LIN {X 0,Y 362.992,Z 430.682,A -85,B 0,C 180,E1 -13571.077,E2 -13571.077} C_VEL
LIN {X 0,Y 362.351,Z 442.962,A -85,B 0,C 180,E1 -13571.921,E2 -13571.921} C_VEL
LIN {X 0,Y 361.612,Z 453.241,A -85,B 0,C 180,E1 -13572.832,E2 -13572.832} C_VEL
LIN {X 0,Y 360.603,Z 463.995,A -85,B 0,C 180,E1 -13574.021,E2 -13574.021} C_VEL
LIN {X 0,Y 359.666,Z 473.198,A -85,B 0,C 180,E1 -13575.285,E2 -13575.285} C_VEL
LIN {X 0,Y 358.837,Z 481.559,A -85,B 0,C 180,E1 -13576.696,E2 -13576.696} C_VEL
LIN {X 0,Y 357.828,Z 489.682,A -85,B 0,C 180,E1 -13578.386,E2 -13578.386} C_VEL
LIN {X 0,Y 356.899,Z 496.795,A -85,B 0,C 180,E1 -13580.247,E2 -13580.247} C_VEL
LIN {X 0,Y 356.33,Z 502.173,A -85,B 0,C 180,E1 -13582.064,E2 -13582.064} C_VEL
LIN {X 0,Y 355.672,Z 506.067,A -85,B 0,C 180,E1 -13583.761,E2 -13583.761} C_VEL
LIN {X 0,Y 355.198,Z 508.939,A -85,B 0,C 180,E1 -13585.461,E2 -13585.461} C_VEL
LIN {X 0,Y 355.19,Z 510.285,A -85,B 0,C 180,E1 -13586.597,E2 -13586.597} C_VEL
LIN {X 0,Y 355.004,Z 511.266,A -85,B 0,C 180,E1 -13587.731,E2 -13587.731} C_VEL
LIN {X 0,Y 355.06,Z 511.847,A -85,B 0,C 180,E1 -13588.866,E2 -13588.866} C_VEL
LIN {X 0,Y 355.04,Z 512.074,A -85,B 0,C 180,E1 -13590,E2 -13590} C_VEL
LIN {X 0,Y 355.06,Z 511.889,A -85,B 0,C 180,E1 -13591.134,E2 -13591.134} C_VEL
LIN {X 0,Y 355.003,Z 511.335,A -85,B 0,C 180,E1 -13592.269,E2 -13592.269} C_VEL
LIN {X 0,Y 355.186,Z 510.382,A -85,B 0,C 180,E1 -13593.403,E2 -13593.403} C_VEL
LIN {X 0,Y 355.187,Z 509.081,A -85,B 0,C 180,E1 -13594.539,E2 -13594.539} C_VEL
LIN {X 0,Y 355.667,Z 506.26,A -85,B 0,C 180,E1 -13596.239,E2 -13596.239} C_VEL
LIN {X 0,Y 356.306,Z 502.433,A -85,B 0,C 180,E1 -13597.936,E2 -13597.936} C_VEL
LIN {X 0,Y 356.836,Z 497.355,A -85,B 0,C 180,E1 -13599.694,E2 -13599.694} C_VEL
LIN {X 0,Y 357.838,Z 490.116,A -85,B 0,C 180,E1 -13601.613,E2 -13601.613} C_VEL
LIN {X 0,Y 358.827,Z 482.089,A -85,B 0,C 180,E1 -13603.305,E2 -13603.305} C_VEL
LIN {X 0,Y 359.677,Z 473.867,A -85,B 0,C 180,E1 -13604.715,E2 -13604.715} C_VEL
LIN {X 0,Y 360.555,Z 464.834,A -85,B 0,C 180,E1 -13605.981,E2 -13605.981} C_VEL
LIN {X 0,Y 361.606,Z 454.324,A -85,B 0,C 180,E1 -13607.161,E2 -13607.161} C_VEL
LIN {X 0,Y 362.403,Z 442.812,A -85,B 0,C 180,E1 -13608.194,E2 -13608.194} C_VEL
LIN {X 0,Y 363.07,Z 431.547,A -85,B 0,C 180,E1 -13608.97,E2 -13608.97} C_VEL
LIN {X 0,Y 363.453,Z 419.23,A -85,B 0,C 180,E1 -13609.595,E2 -13609.595} C_VEL
LIN {X 0,Y 363.551,Z 407.498,A -85,B 0,C 180,E1 -13609.994,E2 -13609.994} C_VEL
LIN {X 0,Y 364.049,Z 361.992,A -85,B 0,C 180,E1 -13610.923,E2 -13610.923} C_VEL
LIN {X 0,Y 364.157,Z 349.57,A -85,B 0,C 180,E1 -13611.175,E2 -13611.175} C_VEL
LIN {X 0,Y 362.973,Z 346.689,A -85,B 0,C 180,E1 -13611.311,E2 -13611.311} C_VEL
LIN {X 0,Y 359.927,Z 343.567,A -85,B 0,C 180,E1 -13611.576,E2 -13611.576} C_VEL
LIN {X 0,Y 352.737,Z 338.216,A -85,B 0,C 180,E1 -13612.177,E2 -13612.177} C_VEL
LIN {X 0,Y 350.859,Z 335.618,A -85,B 0,C 180,E1 -13612.365,E2 -13612.365} C_VEL
LIN {X 0,Y 350.598,Z 335.018,A -85,B 0,C 180,E1 -13612.396,E2 -13612.396} C_VEL
LIN {X 0,Y 347.918,Z 328.96,A -85,B 0,C 180,E1 -13612.76,E2 -13612.76} C_VEL
LIN {X 0,Y 347.766,Z 328.214,A -85,B 0,C 180,E1 -13612.972,E2 -13612.972} C_VEL
LIN {X 0,Y 347.766,Z 328.16,A -85,B 0,C 180,E1 -13615.112,E2 -13615.112} C_VEL
LIN {X 0,Y 347.74,Z 328.146,A -85,B 0,C 180,E1 -13619.015,E2 -13619.015} C_VEL
LIN {X 0,Y 347.734,Z 328.162,A -85,B 0,C 180,E1 -13621.912,E2 -13621.912} C_VEL
LIN {X 0,Y 347.783,Z 328.161,A -85,B 0,C 180,E1 -13625.875,E2 -13625.875} C_VEL
LIN {X 0,Y 347.729,Z 328.162,A -85,B 0,C 180,E1 -13628.795,E2 -13628.795} C_VEL
LIN {X 0,Y 347.737,Z 328.158,A -85,B 0,C 180,E1 -13631.831,E2 -13631.831} C_VEL
LIN {X 0,Y 347.697,Z 328.165,A -85,B 0,C 180,E1 -13635.027,E2 -13635.027} C_VEL
LIN {X 0,Y 347.734,Z 328.162,A -85,B 0,C 180,E1 -13638.399,E2 -13638.399} C_VEL
LIN {X 0,Y 347.758,Z 328.141,A -85,B 0,C 180,E1 -13642.013,E2 -13642.013} C_VEL
LIN {X 0,Y 347.74,Z 328.167,A -85,B 0,C 180,E1 -13645.535,E2 -13645.535} C_VEL
LIN {X 0,Y 347.737,Z 328.145,A -85,B 0,C 180,E1 -13648.299,E2 -13648.299} C_VEL
LIN {X 0,Y 347.735,Z 328.125,A -85,B 0,C 180,E1 -13650.984,E2 -13650.984} C_VEL
LIN {X 0,Y 347.729,Z 328.159,A -85,B 0,C 180,E1 -13653.599,E2 -13653.599} C_VEL
LIN {X 0,Y 347.743,Z 328.169,A -85,B 0,C 180,E1 -13656.158,E2 -13656.158} C_VEL
LIN {X 0,Y 347.774,Z 328.153,A -85,B 0,C 180,E1 -13659.907,E2 -13659.907} C_VEL
LIN {X 0,Y 347.836,Z 328.159,A -85,B 0,C 180,E1 -13662.358,E2 -13662.358} C_VEL
LIN {X 0,Y 347.892,Z 328.133,A -85,B 0,C 180,E1 -13665.97,E2 -13665.97} C_VEL
LIN {X 0,Y 347.887,Z 328.148,A -85,B 0,C 180,E1 -13669.524,E2 -13669.524} C_VEL
LIN {X 0,Y 348.043,Z 328.122,A -85,B 0,C 180,E1 -13673.041,E2 -13673.041} C_VEL
LIN {X 0,Y 348.185,Z 328.108,A -85,B 0,C 180,E1 -13677.686,E2 -13677.686} C_VEL
LIN {X 0,Y 348.133,Z 328.115,A -85,B 0,C 180,E1 -13681.157,E2 -13681.157} C_VEL
LIN {X 0,Y 348.18,Z 328.115,A -85,B 0,C 180,E1 -13682.314,E2 -13682.314} C_VEL
LIN {X 0,Y 348.061,Z 328.118,A -85,B 0,C 180,E1 -13686.959,E2 -13686.959} C_VEL
LIN {X 0,Y 347.885,Z 328.148,A -85,B 0,C 180,E1 -13690.476,E2 -13690.476} C_VEL
LIN {X 0,Y 347.893,Z 328.141,A -85,B 0,C 180,E1 -13694.15,E2 -13694.15} C_VEL
LIN {X 0,Y 347.824,Z 328.148,A -85,B 0,C 180,E1 -13698.259,E2 -13698.259} C_VEL
LIN {X 0,Y 347.761,Z 328.143,A -85,B 0,C 180,E1 -13701.626,E2 -13701.626} C_VEL
LIN {X 0,Y 347.735,Z 328.168,A -85,B 0,C 180,E1 -13705.114,E2 -13705.114} C_VEL
LIN {X 0,Y 347.731,Z 328.154,A -85,B 0,C 180,E1 -13707.701,E2 -13707.701} C_VEL
LIN {X 0,Y 347.734,Z 328.165,A -85,B 0,C 180,E1 -13710.349,E2 -13710.349} C_VEL
LIN {X 0,Y 347.744,Z 328.156,A -85,B 0,C 180,E1 -13714.044,E2 -13714.044} C_VEL
LIN {X 0,Y 347.75,Z 328.167,A -85,B 0,C 180,E1 -13717.322,E2 -13717.322} C_VEL
LIN {X 0,Y 347.693,Z 328.169,A -85,B 0,C 180,E1 -13720.303,E2 -13720.303} C_VEL
LIN {X 0,Y 347.717,Z 328.153,A -85,B 0,C 180,E1 -13723.409,E2 -13723.409} C_VEL
LIN {X 0,Y 347.719,Z 328.156,A -85,B 0,C 180,E1 -13726.688,E2 -13726.688} C_VEL
LIN {X 0,Y 347.698,Z 328.153,A -85,B 0,C 180,E1 -13730.183,E2 -13730.183} C_VEL
LIN {X 0,Y 347.752,Z 328.169,A -85,B 0,C 180,E1 -13732.679,E2 -13732.679} C_VEL
LIN {X 0,Y 347.787,Z 328.368,A -85,B 0,C 180,E1 -13734.104,E2 -13734.104} C_VEL
LIN {X 0,Y 351.19,Z 342.081,A -85,B 0,C 180,E1 -13737.193,E2 -13737.193} C_VEL
LIN {X 0,Y 353.588,Z 353.21,A -85,B 0,C 180,E1 -13739.547,E2 -13739.547} C_VEL
LIN {X 0,Y 353.93,Z 356.668,A -85,B 0,C 180,E1 -13740.237,E2 -13740.237} C_VEL
LIN {X 0,Y 352.145,Z 373.363,A -85,B 0,C 180,E1 -13743.318,E2 -13743.318} C_VEL
LIN {X 0,Y 350.561,Z 389.798,A -85,B 0,C 180,E1 -13746.362,E2 -13746.362} C_VEL
LIN {X 0,Y 350.33,Z 392.943,A -85,B 0,C 180,E1 -13746.907,E2 -13746.907} C_VEL
LIN {X 0,Y 354.663,Z 429.261,A -85,B 0,C 180,E1 -13747.992,E2 -13747.992} C_VEL
LIN {X 0,Y 356.138,Z 446.991,A -85,B 0,C 180,E1 -13748.458,E2 -13748.458} C_VEL
LIN {X 0,Y 355.11,Z 503.797,A -85,B 0,C 180,E1 -13749.623,E2 -13749.623} C_VEL
LIN {X 0,Y 354.371,Z 517.053,A -85,B 0,C 180,E1 -13750.108,E2 -13750.108} C_VEL
LIN {X 0,Y 353.326,Z 530.374,A -85,B 0,C 180,E1 -13750.841,E2 -13750.841} C_VEL
LIN {X 0,Y 352.153,Z 541.578,A -85,B 0,C 180,E1 -13751.68,E2 -13751.68} C_VEL
LIN {X 0,Y 350.865,Z 553.276,A -85,B 0,C 180,E1 -13752.816,E2 -13752.816} C_VEL
LIN {X 0,Y 349.598,Z 562.733,A -85,B 0,C 180,E1 -13753.954,E2 -13753.954} C_VEL
LIN {X 0,Y 348.543,Z 572.718,A -85,B 0,C 180,E1 -13755.437,E2 -13755.437} C_VEL
LIN {X 0,Y 347.821,Z 580.554,A -85,B 0,C 180,E1 -13756.861,E2 -13756.861} C_VEL
LIN {X 0,Y 347.145,Z 588.445,A -85,B 0,C 180,E1 -13758.616,E2 -13758.616} C_VEL
LIN {X 0,Y 346.761,Z 595.768,A -85,B 0,C 180,E1 -13760.669,E2 -13760.669} C_VEL
LIN {X 0,Y 346.754,Z 600.683,A -85,B 0,C 180,E1 -13762.43,E2 -13762.43} C_VEL
LIN {X 0,Y 346.887,Z 604.461,A -85,B 0,C 180,E1 -13764.186,E2 -13764.186} C_VEL
LIN {X 0,Y 347.068,Z 606.426,A -85,B 0,C 180,E1 -13765.354,E2 -13765.354} C_VEL
LIN {X 0,Y 347.192,Z 607.899,A -85,B 0,C 180,E1 -13766.519,E2 -13766.519} C_VEL
LIN {X 0,Y 347.624,Z 609.63,A -85,B 0,C 180,E1 -13768.842,E2 -13768.842} C_VEL
LIN {X 0,Y 347.7,Z 609.864,A -85,B 0,C 180,E1 -13770,E2 -13770} C_VEL
LIN {X 0,Y 347.624,Z 609.626,A -85,B 0,C 180,E1 -13771.158,E2 -13771.158} C_VEL
LIN {X 0,Y 347.197,Z 607.891,A -85,B 0,C 180,E1 -13773.481,E2 -13773.481} C_VEL
LIN {X 0,Y 347.081,Z 606.414,A -85,B 0,C 180,E1 -13774.646,E2 -13774.646} C_VEL
LIN {X 0,Y 346.825,Z 602.403,A -85,B 0,C 180,E1 -13776.817,E2 -13776.817} C_VEL
LIN {X 0,Y 346.717,Z 597.492,A -85,B 0,C 180,E1 -13778.744,E2 -13778.744} C_VEL
LIN {X 0,Y 346.905,Z 591.759,A -85,B 0,C 180,E1 -13780.505,E2 -13780.505} C_VEL
LIN {X 0,Y 347.4,Z 584.652,A -85,B 0,C 180,E1 -13782.264,E2 -13782.264} C_VEL
LIN {X 0,Y 348.243,Z 575.809,A -85,B 0,C 180,E1 -13784.015,E2 -13784.015} C_VEL
LIN {X 0,Y 349.218,Z 566.789,A -85,B 0,C 180,E1 -13785.465,E2 -13785.465} C_VEL
LIN {X 0,Y 350.173,Z 558.113,A -85,B 0,C 180,E1 -13786.618,E2 -13786.618} C_VEL
LIN {X 0,Y 351.6,Z 546.178,A -85,B 0,C 180,E1 -13787.898,E2 -13787.898} C_VEL
LIN {X 0,Y 352.942,Z 534.199,A -85,B 0,C 180,E1 -13788.879,E2 -13788.879} C_VEL
LIN {X 0,Y 354.035,Z 521.753,A -85,B 0,C 180,E1 -13789.647,E2 -13789.647} C_VEL
LIN {X 0,Y 354.852,Z 508.968,A -85,B 0,C 180,E1 -13790.203,E2 -13790.203} C_VEL
LIN {X 0,Y 355.273,Z 495.52,A -85,B 0,C 180,E1 -13790.556,E2 -13790.556} C_VEL
LIN {X 0,Y 356.062,Z 445.027,A -85,B 0,C 180,E1 -13791.573,E2 -13791.573} C_VEL
LIN {X 0,Y 352.693,Z 412.041,A -85,B 0,C 180,E1 -13792.484,E2 -13792.484} C_VEL
LIN {X 0,Y 350.299,Z 393.033,A -85,B 0,C 180,E1 -13793.07,E2 -13793.07} C_VEL
LIN {X 0,Y 351.825,Z 376.583,A -85,B 0,C 180,E1 -13796.069,E2 -13796.069} C_VEL
LIN {X 0,Y 353.939,Z 356.577,A -85,B 0,C 180,E1 -13799.762,E2 -13799.762} C_VEL
LIN {X 0,Y 352.955,Z 349.961,A -85,B 0,C 180,E1 -13801.106,E2 -13801.106} C_VEL
LIN {X 0,Y 350.046,Z 337.188,A -85,B 0,C 180,E1 -13803.858,E2 -13803.858} C_VEL
LIN {X 0,Y 347.794,Z 328.272,A -85,B 0,C 180,E1 -13805.916,E2 -13805.916} C_VEL
LIN {X 0,Y 347.728,Z 328.154,A -85,B 0,C 180,E1 -13808.795,E2 -13808.795} C_VEL
LIN {X 0,Y 347.737,Z 328.172,A -85,B 0,C 180,E1 -13811.831,E2 -13811.831} C_VEL
LIN {X 0,Y 347.695,Z 328.141,A -85,B 0,C 180,E1 -13815.027,E2 -13815.027} C_VEL
LIN {X 0,Y 347.736,Z 328.171,A -85,B 0,C 180,E1 -13818.399,E2 -13818.399} C_VEL
LIN {X 0,Y 347.757,Z 328.115,A -85,B 0,C 180,E1 -13822.014,E2 -13822.014} C_VEL
LIN {X 0,Y 347.738,Z 328.147,A -85,B 0,C 180,E1 -13825.535,E2 -13825.535} C_VEL
LIN {X 0,Y 347.74,Z 328.169,A -85,B 0,C 180,E1 -13828.3,E2 -13828.3} C_VEL
LIN {X 0,Y 347.74,Z 328.151,A -85,B 0,C 180,E1 -13830.984,E2 -13830.984} C_VEL
LIN {X 0,Y 347.74,Z 328.162,A -85,B 0,C 180,E1 -13833.6,E2 -13833.6} C_VEL
LIN {X 0,Y 347.746,Z 328.164,A -85,B 0,C 180,E1 -13836.159,E2 -13836.159} C_VEL
LIN {X 0,Y 347.799,Z 328.135,A -85,B 0,C 180,E1 -13839.908,E2 -13839.908} C_VEL
LIN {X 0,Y 347.861,Z 328.152,A -85,B 0,C 180,E1 -13842.359,E2 -13842.359} C_VEL
LIN {X 0,Y 347.892,Z 328.139,A -85,B 0,C 180,E1 -13845.971,E2 -13845.971} C_VEL
LIN {X 0,Y 347.888,Z 328.148,A -85,B 0,C 180,E1 -13849.524,E2 -13849.524} C_VEL
LIN {X 0,Y 348.065,Z 328.118,A -85,B 0,C 180,E1 -13853.042,E2 -13853.042} C_VEL
LIN {X 0,Y 348.181,Z 328.116,A -85,B 0,C 180,E1 -13857.686,E2 -13857.686} C_VEL
LIN {X 0,Y 348.109,Z 328.105,A -85,B 0,C 180,E1 -13861.157,E2 -13861.157} C_VEL
LIN {X 0,Y 348.185,Z 328.108,A -85,B 0,C 180,E1 -13862.314,E2 -13862.314} C_VEL
LIN {X 0,Y 348.045,Z 328.121,A -85,B 0,C 180,E1 -13866.959,E2 -13866.959} C_VEL
LIN {X 0,Y 347.889,Z 328.147,A -85,B 0,C 180,E1 -13870.476,E2 -13870.476} C_VEL
LIN {X 0,Y 347.893,Z 328.132,A -85,B 0,C 180,E1 -13874.15,E2 -13874.15} C_VEL
LIN {X 0,Y 347.824,Z 328.156,A -85,B 0,C 180,E1 -13878.26,E2 -13878.26} C_VEL
LIN {X 0,Y 347.758,Z 328.156,A -85,B 0,C 180,E1 -13881.625,E2 -13881.625} C_VEL
LIN {X 0,Y 347.732,Z 328.17,A -85,B 0,C 180,E1 -13885.115,E2 -13885.115} C_VEL
LIN {X 0,Y 347.719,Z 328.142,A -85,B 0,C 180,E1 -13887.702,E2 -13887.702} C_VEL
LIN {X 0,Y 347.73,Z 328.128,A -85,B 0,C 180,E1 -13890.35,E2 -13890.35} C_VEL
LIN {X 0,Y 347.744,Z 328.168,A -85,B 0,C 180,E1 -13894.044,E2 -13894.044} C_VEL
LIN {X 0,Y 347.752,Z 328.149,A -85,B 0,C 180,E1 -13897.322,E2 -13897.322} C_VEL
LIN {X 0,Y 347.692,Z 328.149,A -85,B 0,C 180,E1 -13900.303,E2 -13900.303} C_VEL
LIN {X 0,Y 347.717,Z 328.175,A -85,B 0,C 180,E1 -13903.409,E2 -13903.409} C_VEL
LIN {X 0,Y 347.719,Z 328.147,A -85,B 0,C 180,E1 -13906.688,E2 -13906.688} C_VEL
LIN {X 0,Y 347.698,Z 328.173,A -85,B 0,C 180,E1 -13910.183,E2 -13910.183} C_VEL
LIN {X 0,Y 347.753,Z 328.149,A -85,B 0,C 180,E1 -13912.679,E2 -13912.679} C_VEL
LIN {X 0,Y 347.747,Z 328.165,A -85,B 0,C 180,E1 -13915.957,E2 -13915.957} C_VEL
LIN {X 0,Y 347.737,Z 328.17,A -85,B 0,C 180,E1 -13919.652,E2 -13919.652} C_VEL
LIN {X 0,Y 347.737,Z 328.137,A -85,B 0,C 180,E1 -13923.601,E2 -13923.601} C_VEL
LIN {X 0,Y 347.776,Z 328.152,A -85,B 0,C 180,E1 -13926.95,E2 -13926.95} C_VEL
LIN {X 0,Y 347.869,Z 328.637,A -85,B 0,C 180,E1 -13927.29,E2 -13927.29} C_VEL
LIN {X 0,Y 348.478,Z 330.441,A -85,B 0,C 180,E1 -13927.462,E2 -13927.462} C_VEL
LIN {X 0,Y 357.121,Z 350.166,A -85,B 0,C 180,E1 -13928.486,E2 -13928.486} C_VEL
LIN {X 0,Y 357.672,Z 351.901,A -85,B 0,C 180,E1 -13928.559,E2 -13928.559} C_VEL
LIN {X 0,Y 356.92,Z 405.575,A -85,B 0,C 180,E1 -13929.653,E2 -13929.653} C_VEL
LIN {X 0,Y 356.833,Z 417.606,A -85,B 0,C 180,E1 -13930.026,E2 -13930.026} C_VEL
LIN {X 0,Y 356.39,Z 430.387,A -85,B 0,C 180,E1 -13930.638,E2 -13930.638} C_VEL
LIN {X 0,Y 355.786,Z 442.728,A -85,B 0,C 180,E1 -13931.472,E2 -13931.472} C_VEL
LIN {X 0,Y 354.898,Z 454.227,A -85,B 0,C 180,E1 -13932.497,E2 -13932.497} C_VEL
LIN {X 0,Y 353.851,Z 464.977,A -85,B 0,C 180,E1 -13933.708,E2 -13933.708} C_VEL
LIN {X 0,Y 352.872,Z 474.18,A -85,B 0,C 180,E1 -13934.995,E2 -13934.995} C_VEL
LIN {X 0,Y 352.001,Z 482.54,A -85,B 0,C 180,E1 -13936.432,E2 -13936.432} C_VEL
LIN {X 0,Y 350.947,Z 490.662,A -85,B 0,C 180,E1 -13938.155,E2 -13938.155} C_VEL
LIN {X 0,Y 349.974,Z 497.774,A -85,B 0,C 180,E1 -13940.052,E2 -13940.052} C_VEL
LIN {X 0,Y 349.371,Z 503.152,A -85,B 0,C 180,E1 -13941.905,E2 -13941.905} C_VEL
LIN {X 0,Y 348.687,Z 507.046,A -85,B 0,C 180,E1 -13943.635,E2 -13943.635} C_VEL
LIN {X 0,Y 348.188,Z 509.919,A -85,B 0,C 180,E1 -13945.369,E2 -13945.369} C_VEL
LIN {X 0,Y 348.173,Z 511.264,A -85,B 0,C 180,E1 -13946.528,E2 -13946.528} C_VEL
LIN {X 0,Y 347.982,Z 512.244,A -85,B 0,C 180,E1 -13947.685,E2 -13947.685} C_VEL
LIN {X 0,Y 348.035,Z 512.825,A -85,B 0,C 180,E1 -13948.843,E2 -13948.843} C_VEL
LIN {X 0,Y 348.014,Z 513.052,A -85,B 0,C 180,E1 -13950,E2 -13950} C_VEL
LIN {X 0,Y 348.035,Z 512.867,A -85,B 0,C 180,E1 -13951.157,E2 -13951.157} C_VEL
LIN {X 0,Y 347.981,Z 512.313,A -85,B 0,C 180,E1 -13952.315,E2 -13952.315} C_VEL
LIN {X 0,Y 348.17,Z 511.36,A -85,B 0,C 180,E1 -13953.472,E2 -13953.472} C_VEL
LIN {X 0,Y 348.178,Z 510.059,A -85,B 0,C 180,E1 -13954.631,E2 -13954.631} C_VEL
LIN {X 0,Y 348.682,Z 507.237,A -85,B 0,C 180,E1 -13956.365,E2 -13956.365} C_VEL
LIN {X 0,Y 349.346,Z 503.41,A -85,B 0,C 180,E1 -13958.095,E2 -13958.095} C_VEL
LIN {X 0,Y 349.91,Z 498.331,A -85,B 0,C 180,E1 -13959.888,E2 -13959.888} C_VEL
LIN {X 0,Y 350.957,Z 491.092,A -85,B 0,C 180,E1 -13961.844,E2 -13961.844} C_VEL
LIN {X 0,Y 351.991,Z 483.064,A -85,B 0,C 180,E1 -13963.568,E2 -13963.568} C_VEL
LIN {X 0,Y 352.881,Z 474.842,A -85,B 0,C 180,E1 -13965.005,E2 -13965.005} C_VEL
LIN {X 0,Y 353.804,Z 465.808,A -85,B 0,C 180,E1 -13966.295,E2 -13966.295} C_VEL
LIN {X 0,Y 354.899,Z 455.297,A -85,B 0,C 180,E1 -13967.495,E2 -13967.495} C_VEL
LIN {X 0,Y 355.734,Z 443.784,A -85,B 0,C 180,E1 -13968.548,E2 -13968.548} C_VEL
LIN {X 0,Y 356.424,Z 432.518,A -85,B 0,C 180,E1 -13969.338,E2 -13969.338} C_VEL
LIN {X 0,Y 356.827,Z 420.234,A -85,B 0,C 180,E1 -13969.972,E2 -13969.972} C_VEL
LIN {X 0,Y 356.93,Z 408.58,A -85,B 0,C 180,E1 -13970.378,E2 -13970.378} C_VEL
LIN {X 0,Y 357.404,Z 364.617,A -85,B 0,C 180,E1 -13971.295,E2 -13971.295} C_VEL
LIN {X 0,Y 357.492,Z 351.015,A -85,B 0,C 180,E1 -13971.579,E2 -13971.579} C_VEL
LIN {X 0,Y 350.598,Z 335.018,A -85,B 0,C 180,E1 -13972.396,E2 -13972.396} C_VEL
LIN {X 0,Y 349.299,Z 332.491,A -85,B 0,C 180,E1 -13972.637,E2 -13972.637} C_VEL
LIN {X 0,Y 347.42,Z 330.284,A -85,B 0,C 180,E1 -13973.132,E2 -13973.132} C_VEL
LIN {X 0,Y 345.747,Z 329.119,A -85,B 0,C 180,E1 -13973.682,E2 -13973.682} C_VEL
LIN {X 0,Y 343.894,Z 328.649,A -85,B 0,C 180,E1 -13974.45,E2 -13974.45} C_VEL
LIN {X 0,Y 341.749,Z 328.893,A -85,B 0,C 180,E1 -13975.684,E2 -13975.684} C_VEL
LIN {X 0,Y 340.787,Z 329.007,A -85,B 0,C 180,E1 -13976.777,E2 -13976.777} C_VEL
LIN {X 0,Y 340.699,Z 329.005,A -85,B 0,C 180,E1 -13977.146,E2 -13977.146} C_VEL
LIN {X 0,Y 340.689,Z 329.047,A -85,B 0,C 180,E1 -13981.045,E2 -13981.045} C_VEL
LIN {X 0,Y 340.714,Z 329.044,A -85,B 0,C 180,E1 -13985.279,E2 -13985.279} C_VEL
LIN {X 0,Y 340.691,Z 329.034,A -85,B 0,C 180,E1 -13988.382,E2 -13988.382} C_VEL
LIN {X 0,Y 340.688,Z 329.032,A -85,B 0,C 180,E1 -13992.043,E2 -13992.043} C_VEL
LIN {X 0,Y 340.646,Z 329.052,A -85,B 0,C 180,E1 -13996.227,E2 -13996.227} C_VEL
LIN {X 0,Y 340.665,Z 329.038,A -85,B 0,C 180,E1 -13998.687,E2 -13998.687} C_VEL
LIN {X 0,Y 340.715,Z 329.015,A -85,B 0,C 180,E1 -14001.77,E2 -14001.77} C_VEL
LIN {X 0,Y 340.719,Z 329.042,A -85,B 0,C 180,E1 -14005.595,E2 -14005.595} C_VEL
LIN {X 0,Y 340.686,Z 329.014,A -85,B 0,C 180,E1 -14008.954,E2 -14008.954} C_VEL
LIN {X 0,Y 340.705,Z 329.025,A -85,B 0,C 180,E1 -14013.011,E2 -14013.011} C_VEL
LIN {X 0,Y 340.695,Z 329.043,A -85,B 0,C 180,E1 -14016.925,E2 -14016.925} C_VEL
LIN {X 0,Y 340.718,Z 329.04,A -85,B 0,C 180,E1 -14020.729,E2 -14020.729} C_VEL
LIN {X 0,Y 340.809,Z 329.02,A -85,B 0,C 180,E1 -14024.45,E2 -14024.45} C_VEL
LIN {X 0,Y 340.841,Z 329.026,A -85,B 0,C 180,E1 -14028.1,E2 -14028.1} C_VEL
LIN {X 0,Y 340.974,Z 328.998,A -85,B 0,C 180,E1 -14031.704,E2 -14031.704} C_VEL
LIN {X 0,Y 341.003,Z 329.002,A -85,B 0,C 180,E1 -14034.085,E2 -14034.085} C_VEL
LIN {X 0,Y 341.122,Z 328.987,A -85,B 0,C 180,E1 -14037.638,E2 -14037.638} C_VEL
LIN {X 0,Y 341.102,Z 328.991,A -85,B 0,C 180,E1 -14041.181,E2 -14041.181} C_VEL
LIN {X 0,Y 341.117,Z 328.995,A -85,B 0,C 180,E1 -14042.362,E2 -14042.362} C_VEL
LIN {X 0,Y 341.017,Z 328.991,A -85,B 0,C 180,E1 -14045.914,E2 -14045.914} C_VEL
LIN {X 0,Y 340.958,Z 329.011,A -85,B 0,C 180,E1 -14048.356,E2 -14048.356} C_VEL
LIN {X 0,Y 340.839,Z 329.018,A -85,B 0,C 180,E1 -14051.9,E2 -14051.9} C_VEL
LIN {X 0,Y 340.811,Z 329.03,A -85,B 0,C 180,E1 -14055.55,E2 -14055.55} C_VEL
LIN {X 0,Y 340.756,Z 329.021,A -85,B 0,C 180,E1 -14059.269,E2 -14059.269} C_VEL
LIN {X 0,Y 340.7,Z 329.04,A -85,B 0,C 180,E1 -14063.075,E2 -14063.075} C_VEL
LIN {X 0,Y 340.714,Z 329.033,A -85,B 0,C 180,E1 -14066.988,E2 -14066.988} C_VEL
LIN {X 0,Y 340.689,Z 329.046,A -85,B 0,C 180,E1 -14071.046,E2 -14071.046} C_VEL
LIN {X 0,Y 340.711,Z 329.034,A -85,B 0,C 180,E1 -14075.28,E2 -14075.28} C_VEL
LIN {X 0,Y 340.688,Z 329.04,A -85,B 0,C 180,E1 -14078.383,E2 -14078.383} C_VEL
LIN {X 0,Y 340.688,Z 329.046,A -85,B 0,C 180,E1 -14082.045,E2 -14082.045} C_VEL
LIN {X 0,Y 340.645,Z 329.027,A -85,B 0,C 180,E1 -14086.228,E2 -14086.228} C_VEL
LIN {X 0,Y 340.665,Z 329.047,A -85,B 0,C 180,E1 -14088.688,E2 -14088.688} C_VEL
LIN {X 0,Y 340.716,Z 329.034,A -85,B 0,C 180,E1 -14091.771,E2 -14091.771} C_VEL
LIN {X 0,Y 340.751,Z 329.237,A -85,B 0,C 180,E1 -14093.643,E2 -14093.643} C_VEL
LIN {X 0,Y 344.217,Z 343.037,A -85,B 0,C 180,E1 -14096.837,E2 -14096.837} C_VEL
LIN {X 0,Y 346.893,Z 355.659,A -85,B 0,C 180,E1 -14099.57,E2 -14099.57} C_VEL
LIN {X 0,Y 346.885,Z 359.98,A -85,B 0,C 180,E1 -14100.42,E2 -14100.42} C_VEL
LIN {X 0,Y 344.706,Z 379.664,A -85,B 0,C 180,E1 -14104.136,E2 -14104.136} C_VEL
LIN {X 0,Y 343.495,Z 391.959,A -85,B 0,C 180,E1 -14106.422,E2 -14106.422} C_VEL
LIN {X 0,Y 347.206,Z 422.394,A -85,B 0,C 180,E1 -14107.368,E2 -14107.368} C_VEL
LIN {X 0,Y 349.514,Z 447.189,A -85,B 0,C 180,E1 -14108.054,E2 -14108.054} C_VEL
LIN {X 0,Y 348.469,Z 502.823,A -85,B 0,C 180,E1 -14109.217,E2 -14109.217} C_VEL
LIN {X 0,Y 347.669,Z 516.069,A -85,B 0,C 180,E1 -14109.708,E2 -14109.708} C_VEL
LIN {X 0,Y 346.632,Z 529.393,A -85,B 0,C 180,E1 -14110.456,E2 -14110.456} C_VEL
LIN {X 0,Y 345.41,Z 540.593,A -85,B 0,C 180,E1 -14111.309,E2 -14111.309} C_VEL
LIN {X 0,Y 343.975,Z 552.276,A -85,B 0,C 180,E1 -14112.461,E2 -14112.461} C_VEL
LIN {X 0,Y 342.602,Z 562.827,A -85,B 0,C 180,E1 -14113.77,E2 -14113.77} C_VEL
LIN {X 0,Y 341.489,Z 572.707,A -85,B 0,C 180,E1 -14115.304,E2 -14115.304} C_VEL
LIN {X 0,Y 340.665,Z 580.966,A -85,B 0,C 180,E1 -14116.884,E2 -14116.884} C_VEL
LIN {X 0,Y 340.053,Z 588.605,A -85,B 0,C 180,E1 -14118.677,E2 -14118.677} C_VEL
LIN {X 0,Y 339.698,Z 594.773,A -85,B 0,C 180,E1 -14120.473,E2 -14120.473} C_VEL
LIN {X 0,Y 339.668,Z 599.689,A -85,B 0,C 180,E1 -14122.271,E2 -14122.271} C_VEL
LIN {X 0,Y 339.82,Z 603.473,A -85,B 0,C 180,E1 -14124.065,E2 -14124.065} C_VEL
LIN {X 0,Y 340.006,Z 605.441,A -85,B 0,C 180,E1 -14125.257,E2 -14125.257} C_VEL
LIN {X 0,Y 340.142,Z 606.916,A -85,B 0,C 180,E1 -14126.446,E2 -14126.446} C_VEL
LIN {X 0,Y 340.588,Z 608.651,A -85,B 0,C 180,E1 -14128.818,E2 -14128.818} C_VEL
LIN {X 0,Y 340.673,Z 608.886,A -85,B 0,C 180,E1 -14130,E2 -14130} C_VEL
LIN {X 0,Y 340.589,Z 608.646,A -85,B 0,C 180,E1 -14131.182,E2 -14131.182} C_VEL
LIN {X 0,Y 340.147,Z 606.908,A -85,B 0,C 180,E1 -14133.554,E2 -14133.554} C_VEL
LIN {X 0,Y 340.019,Z 605.428,A -85,B 0,C 180,E1 -14134.742,E2 -14134.742} C_VEL
LIN {X 0,Y 339.768,Z 601.66,A -85,B 0,C 180,E1 -14136.846,E2 -14136.846} C_VEL
LIN {X 0,Y 339.659,Z 596.497,A -85,B 0,C 180,E1 -14138.927,E2 -14138.927} C_VEL
LIN {X 0,Y 339.853,Z 590.759,A -85,B 0,C 180,E1 -14140.726,E2 -14140.726} C_VEL
LIN {X 0,Y 340.392,Z 583.652,A -85,B 0,C 180,E1 -14142.52,E2 -14142.52} C_VEL
LIN {X 0,Y 341.15,Z 576.441,A -85,B 0,C 180,E1 -14144.008,E2 -14144.008} C_VEL
LIN {X 0,Y 342.1,Z 567.774,A -85,B 0,C 180,E1 -14145.49,E2 -14145.49} C_VEL
LIN {X 0,Y 343.186,Z 558.304,A -85,B 0,C 180,E1 -14146.813,E2 -14146.813} C_VEL
LIN {X 0,Y 344.644,Z 546.624,A -85,B 0,C 180,E1 -14148.118,E2 -14148.118} C_VEL
LIN {X 0,Y 345.989,Z 535.151,A -85,B 0,C 180,E1 -14149.119,E2 -14149.119} C_VEL
LIN {X 0,Y 347.136,Z 523.37,A -85,B 0,C 180,E1 -14149.9,E2 -14149.9} C_VEL
LIN {X 0,Y 348.108,Z 509.815,A -85,B 0,C 180,E1 -14150.535,E2 -14150.535} C_VEL
LIN {X 0,Y 348.566,Z 497.879,A -85,B 0,C 180,E1 -14150.893,E2 -14150.893} C_VEL
LIN {X 0,Y 349.454,Z 446.191,A -85,B 0,C 180,E1 -14151.955,E2 -14151.955} C_VEL
LIN {X 0,Y 346.359,Z 415.148,A -85,B 0,C 180,E1 -14152.829,E2 -14152.829} C_VEL
LIN {X 0,Y 343.5,Z 391.867,A -85,B 0,C 180,E1 -14153.567,E2 -14153.567} C_VEL
LIN {X 0,Y 345.846,Z 368.961,A -85,B 0,C 180,E1 -14157.864,E2 -14157.864} C_VEL
LIN {X 0,Y 347.043,Z 357.198,A -85,B 0,C 180,E1 -14160.097,E2 -14160.097} C_VEL
LIN {X 0,Y 345.434,Z 348.514,A -85,B 0,C 180,E1 -14161.936,E2 -14161.936} C_VEL
LIN {X 0,Y 342.083,Z 334.35,A -85,B 0,C 180,E1 -14165.117,E2 -14165.117} C_VEL
LIN {X 0,Y 340.72,Z 329.123,A -85,B 0,C 180,E1 -14166.405,E2 -14166.405} C_VEL
LIN {X 0,Y 340.652,Z 329.031,A -85,B 0,C 180,E1 -14169.758,E2 -14169.758} C_VEL
LIN {X 0,Y 340.668,Z 329.043,A -85,B 0,C 180,E1 -14172.904,E2 -14172.904} C_VEL
LIN {X 0,Y 340.669,Z 329.044,A -85,B 0,C 180,E1 -14177.094,E2 -14177.094} C_VEL
LIN {X 0,Y 340.651,Z 329.038,A -85,B 0,C 180,E1 -14180.241,E2 -14180.241} C_VEL
LIN {X 0,Y 340.701,Z 328.988,A -85,B 0,C 180,E1 -14183.56,E2 -14183.56} C_VEL
LIN {X 0,Y 340.688,Z 329.033,A -85,B 0,C 180,E1 -14186.153,E2 -14186.153} C_VEL
LIN {X 0,Y 340.716,Z 329.032,A -85,B 0,C 180,E1 -14190.034,E2 -14190.034} C_VEL
LIN {X 0,Y 340.714,Z 329.034,A -85,B 0,C 180,E1 -14193.012,E2 -14193.012} C_VEL
LIN {X 0,Y 340.7,Z 329.039,A -85,B 0,C 180,E1 -14196.925,E2 -14196.925} C_VEL
LIN {X 0,Y 340.782,Z 329.019,A -85,B 0,C 180,E1 -14200.733,E2 -14200.733} C_VEL
LIN {X 0,Y 340.78,Z 329.034,A -85,B 0,C 180,E1 -14203.218,E2 -14203.218} C_VEL
LIN {X 0,Y 340.837,Z 329.013,A -85,B 0,C 180,E1 -14206.89,E2 -14206.89} C_VEL
LIN {X 0,Y 340.875,Z 329.022,A -85,B 0,C 180,E1 -14210.506,E2 -14210.506} C_VEL
LIN {X 0,Y 341.018,Z 328.992,A -85,B 0,C 180,E1 -14214.086,E2 -14214.086} C_VEL
LIN {X 0,Y 341.118,Z 328.996,A -85,B 0,C 180,E1 -14217.638,E2 -14217.638} C_VEL
LIN {X 0,Y 341.081,Z 328.98,A -85,B 0,C 180,E1 -14221.181,E2 -14221.181} C_VEL
LIN {X 0,Y 341.123,Z 328.987,A -85,B 0,C 180,E1 -14222.362,E2 -14222.362} C_VEL
LIN {X 0,Y 340.993,Z 328.997,A -85,B 0,C 180,E1 -14227.104,E2 -14227.104} C_VEL
LIN {X 0,Y 340.841,Z 329.024,A -85,B 0,C 180,E1 -14230.695,E2 -14230.695} C_VEL
LIN {X 0,Y 340.858,Z 329.008,A -85,B 0,C 180,E1 -14234.325,E2 -14234.325} C_VEL
LIN {X 0,Y 340.781,Z 329.033,A -85,B 0,C 180,E1 -14238.441,E2 -14238.441} C_VEL
LIN {X 0,Y 340.713,Z 329.035,A -85,B 0,C 180,E1 -14241.842,E2 -14241.842} C_VEL
LIN {X 0,Y 340.665,Z 329.043,A -85,B 0,C 180,E1 -14245.673,E2 -14245.673} C_VEL
LIN {X 0,Y 340.67,Z 329.012,A -85,B 0,C 180,E1 -14248.326,E2 -14248.326} C_VEL
LIN {X 0,Y 340.686,Z 329.014,A -85,B 0,C 180,E1 -14251.046,E2 -14251.046} C_VEL
LIN {X 0,Y 340.713,Z 329.046,A -85,B 0,C 180,E1 -14255.28,E2 -14255.28} C_VEL
LIN {X 0,Y 340.689,Z 329.017,A -85,B 0,C 180,E1 -14258.383,E2 -14258.383} C_VEL
LIN {X 0,Y 340.687,Z 329.045,A -85,B 0,C 180,E1 -14262.044,E2 -14262.044} C_VEL
LIN {X 0,Y 340.646,Z 329.029,A -85,B 0,C 180,E1 -14266.228,E2 -14266.228} C_VEL
LIN {X 0,Y 340.665,Z 329.043,A -85,B 0,C 180,E1 -14268.688,E2 -14268.688} C_VEL
LIN {X 0,Y 340.716,Z 329.03,A -85,B 0,C 180,E1 -14271.771,E2 -14271.771} C_VEL
LIN {X 0,Y 340.721,Z 329.043,A -85,B 0,C 180,E1 -14275.596,E2 -14275.596} C_VEL
LIN {X 0,Y 340.692,Z 329.046,A -85,B 0,C 180,E1 -14278.955,E2 -14278.955} C_VEL
LIN {X 0,Y 340.71,Z 329.006,A -85,B 0,C 180,E1 -14283.012,E2 -14283.012} C_VEL
LIN {X 0,Y 340.727,Z 329.147,A -85,B 0,C 180,E1 -14286.646,E2 -14286.646} C_VEL
LIN {X 0,Y 340.923,Z 330.03,A -85,B 0,C 180,E1 -14286.871,E2 -14286.871} C_VEL
LIN {X 0,Y 350.239,Z 351.142,A -85,B 0,C 180,E1 -14288.04,E2 -14288.04} C_VEL
LIN {X 0,Y 350.966,Z 352.922,A -85,B 0,C 180,E1 -14288.129,E2 -14288.129} C_VEL
LIN {X 0,Y 350.257,Z 411.138,A -85,B 0,C 180,E1 -14289.366,E2 -14289.366} C_VEL
LIN {X 0,Y 350.016,Z 424.108,A -85,B 0,C 180,E1 -14289.869,E2 -14289.869} C_VEL
LIN {X 0,Y 349.531,Z 437.16,A -85,B 0,C 180,E1 -14290.625,E2 -14290.625} C_VEL
LIN {X 0,Y 348.807,Z 448.763,A -85,B 0,C 180,E1 -14291.534,E2 -14291.534} C_VEL
LIN {X 0,Y 347.704,Z 459.939,A -85,B 0,C 180,E1 -14292.655,E2 -14292.655} C_VEL
LIN {X 0,Y 346.627,Z 470.27,A -85,B 0,C 180,E1 -14293.964,E2 -14293.964} C_VEL
LIN {X 0,Y 345.709,Z 478.688,A -85,B 0,C 180,E1 -14295.279,E2 -14295.279} C_VEL
LIN {X 0,Y 344.723,Z 486.439,A -85,B 0,C 180,E1 -14296.741,E2 -14296.741} C_VEL
LIN {X 0,Y 343.72,Z 494.11,A -85,B 0,C 180,E1 -14298.531,E2 -14298.531} C_VEL
LIN {X 0,Y 342.936,Z 499.862,A -85,B 0,C 180,E1 -14300.205,E2 -14300.205} C_VEL
LIN {X 0,Y 342.415,Z 504.131,A -85,B 0,C 180,E1 -14301.74,E2 -14301.74} C_VEL
LIN {X 0,Y 341.703,Z 508.025,A -85,B 0,C 180,E1 -14303.505,E2 -14303.505} C_VEL
LIN {X 0,Y 341.18,Z 510.898,A -85,B 0,C 180,E1 -14305.274,E2 -14305.274} C_VEL
LIN {X 0,Y 341.157,Z 512.242,A -85,B 0,C 180,E1 -14306.457,E2 -14306.457} C_VEL
LIN {X 0,Y 340.96,Z 513.222,A -85,B 0,C 180,E1 -14307.637,E2 -14307.637} C_VEL
LIN {X 0,Y 341.009,Z 513.803,A -85,B 0,C 180,E1 -14308.819,E2 -14308.819} C_VEL
LIN {X 0,Y 340.987,Z 514.03,A -85,B 0,C 180,E1 -14310,E2 -14310} C_VEL
LIN {X 0,Y 341.009,Z 513.844,A -85,B 0,C 180,E1 -14311.181,E2 -14311.181} C_VEL
LIN {X 0,Y 340.96,Z 513.29,A -85,B 0,C 180,E1 -14312.363,E2 -14312.363} C_VEL
LIN {X 0,Y 341.153,Z 512.337,A -85,B 0,C 180,E1 -14313.543,E2 -14313.543} C_VEL
LIN {X 0,Y 341.169,Z 511.036,A -85,B 0,C 180,E1 -14314.726,E2 -14314.726} C_VEL
LIN {X 0,Y 341.698,Z 508.214,A -85,B 0,C 180,E1 -14316.495,E2 -14316.495} C_VEL
LIN {X 0,Y 342.39,Z 504.387,A -85,B 0,C 180,E1 -14318.261,E2 -14318.261} C_VEL
LIN {X 0,Y 342.989,Z 499.308,A -85,B 0,C 180,E1 -14320.089,E2 -14320.089} C_VEL
LIN {X 0,Y 344.082,Z 492.068,A -85,B 0,C 180,E1 -14322.085,E2 -14322.085} C_VEL
LIN {X 0,Y 345.162,Z 484.04,A -85,B 0,C 180,E1 -14323.842,E2 -14323.842} C_VEL
LIN {X 0,Y 346.095,Z 475.817,A -85,B 0,C 180,E1 -14325.306,E2 -14325.306} C_VEL
LIN {X 0,Y 347.063,Z 466.782,A -85,B 0,C 180,E1 -14326.62,E2 -14326.62} C_VEL
LIN {X 0,Y 348.198,Z 456.272,A -85,B 0,C 180,E1 -14327.843,E2 -14327.843} C_VEL
LIN {X 0,Y 349.101,Z 444.599,A -85,B 0,C 180,E1 -14328.927,E2 -14328.927} C_VEL
LIN {X 0,Y 349.827,Z 433.15,A -85,B 0,C 180,E1 -14329.74,E2 -14329.74} C_VEL
LIN {X 0,Y 350.223,Z 420.472,A -85,B 0,C 180,E1 -14330.396,E2 -14330.396} C_VEL
LIN {X 0,Y 350.321,Z 410.064,A -85,B 0,C 180,E1 -14330.767,E2 -14330.767} C_VEL
LIN {X 0,Y 350.7,Z 373.077,A -85,B 0,C 180,E1 -14331.56,E2 -14331.56} C_VEL
LIN {X 0,Y 350.939,Z 352.812,A -85,B 0,C 180,E1 -14331.984,E2 -14331.984} C_VEL
LIN {X 0,Y 341.668,Z 331.79,A -85,B 0,C 180,E1 -14333.117,E2 -14333.117} C_VEL
LIN {X 0,Y 340.797,Z 329.564,A -85,B 0,C 180,E1 -14333.309,E2 -14333.309} C_VEL
LIN {X 0,Y 340.735,Z 329.056,A -85,B 0,C 180,E1 -14333.554,E2 -14333.554} C_VEL
LIN {X 0,Y 340.699,Z 329.005,A -85,B 0,C 180,E1 -14337.146,E2 -14337.146} C_VEL
LIN {X 0,Y 339.992,Z 329.1,A -85,B 0,C 180,E1 -14338.133,E2 -14338.133} C_VEL
LIN {X 0,Y 337.108,Z 329.484,A -85,B 0,C 180,E1 -14339.738,E2 -14339.738} C_VEL
LIN {X 0,Y 334.704,Z 329.792,A -85,B 0,C 180,E1 -14341.038,E2 -14341.038} C_VEL
LIN {X 0,Y 333.7,Z 329.908,A -85,B 0,C 180,E1 -14342.044,E2 -14342.044} C_VEL
LIN {X 0,Y 333.631,Z 329.914,A -85,B 0,C 180,E1 -14342.385,E2 -14342.385} C_VEL
LIN {X 0,Y 333.672,Z 329.912,A -85,B 0,C 180,E1 -14346.139,E2 -14346.139} C_VEL
LIN {X 0,Y 333.618,Z 329.926,A -85,B 0,C 180,E1 -14349.196,E2 -14349.196} C_VEL
LIN {X 0,Y 333.623,Z 329.905,A -85,B 0,C 180,E1 -14352.498,E2 -14352.498} C_VEL
LIN {X 0,Y 333.59,Z 329.929,A -85,B 0,C 180,E1 -14355.954,E2 -14355.954} C_VEL
LIN {X 0,Y 333.598,Z 329.911,A -85,B 0,C 180,E1 -14359.324,E2 -14359.324} C_VEL
LIN {X 0,Y 333.659,Z 329.91,A -85,B 0,C 180,E1 -14363.168,E2 -14363.168} C_VEL
LIN {X 0,Y 333.67,Z 329.92,A -85,B 0,C 180,E1 -14365.341,E2 -14365.341} C_VEL
LIN {X 0,Y 333.622,Z 329.902,A -85,B 0,C 180,E1 -14368.221,E2 -14368.221} C_VEL
LIN {X 0,Y 333.623,Z 329.881,A -85,B 0,C 180,E1 -14371.019,E2 -14371.019} C_VEL
LIN {X 0,Y 333.652,Z 329.924,A -85,B 0,C 180,E1 -14374.922,E2 -14374.922} C_VEL
LIN {X 0,Y 333.649,Z 329.91,A -85,B 0,C 180,E1 -14379.017,E2 -14379.017} C_VEL
LIN {X 0,Y 333.734,Z 329.911,A -85,B 0,C 180,E1 -14381.586,E2 -14381.586} C_VEL
LIN {X 0,Y 333.803,Z 329.886,A -85,B 0,C 180,E1 -14385.577,E2 -14385.577} C_VEL
LIN {X 0,Y 333.809,Z 329.902,A -85,B 0,C 180,E1 -14389.077,E2 -14389.077} C_VEL
LIN {X 0,Y 333.947,Z 329.874,A -85,B 0,C 180,E1 -14392.746,E2 -14392.746} C_VEL
LIN {X 0,Y 333.776,Z 329.907,A -85,B 0,C 180,E1 -14395.169,E2 -14395.169} C_VEL
LIN {X 0,Y 334.063,Z 329.867,A -85,B 0,C 180,E1 -14397.588,E2 -14397.588} C_VEL
LIN {X 0,Y 334.07,Z 329.866,A -85,B 0,C 180,E1 -14401.205,E2 -14401.205} C_VEL
LIN {X 0,Y 333.795,Z 329.903,A -85,B 0,C 180,E1 -14403.621,E2 -14403.621} C_VEL
LIN {X 0,Y 333.99,Z 329.865,A -85,B 0,C 180,E1 -14406.039,E2 -14406.039} C_VEL
LIN {X 0,Y 333.812,Z 329.902,A -85,B 0,C 180,E1 -14409.697,E2 -14409.697} C_VEL
LIN {X 0,Y 333.789,Z 329.892,A -85,B 0,C 180,E1 -14413.392,E2 -14413.392} C_VEL
LIN {X 0,Y 333.713,Z 329.912,A -85,B 0,C 180,E1 -14417.148,E2 -14417.148} C_VEL
LIN {X 0,Y 333.682,Z 329.895,A -85,B 0,C 180,E1 -14419.694,E2 -14419.694} C_VEL
LIN {X 0,Y 333.64,Z 329.92,A -85,B 0,C 180,E1 -14423.592,E2 -14423.592} C_VEL
LIN {X 0,Y 333.662,Z 329.905,A -85,B 0,C 180,E1 -14427.606,E2 -14427.606} C_VEL
LIN {X 0,Y 333.652,Z 329.918,A -85,B 0,C 180,E1 -14430.367,E2 -14430.367} C_VEL
LIN {X 0,Y 333.632,Z 329.921,A -85,B 0,C 180,E1 -14433.209,E2 -14433.209} C_VEL
LIN {X 0,Y 333.669,Z 329.917,A -85,B 0,C 180,E1 -14436.14,E2 -14436.14} C_VEL
LIN {X 0,Y 333.597,Z 329.919,A -85,B 0,C 180,E1 -14439.199,E2 -14439.199} C_VEL
LIN {X 0,Y 333.624,Z 329.922,A -85,B 0,C 180,E1 -14442.499,E2 -14442.499} C_VEL
LIN {X 0,Y 333.589,Z 329.901,A -85,B 0,C 180,E1 -14445.955,E2 -14445.955} C_VEL
LIN {X 0,Y 333.599,Z 329.915,A -85,B 0,C 180,E1 -14449.325,E2 -14449.325} C_VEL
LIN {X 0,Y 333.694,Z 330.113,A -85,B 0,C 180,E1 -14453.161,E2 -14453.161} C_VEL
LIN {X 0,Y 337.213,Z 344.028,A -85,B 0,C 180,E1 -14456.476,E2 -14456.476} C_VEL
LIN {X 0,Y 339.841,Z 356.343,A -85,B 0,C 180,E1 -14459.215,E2 -14459.215} C_VEL
LIN {X 0,Y 340.157,Z 359.786,A -85,B 0,C 180,E1 -14459.933,E2 -14459.933} C_VEL
LIN {X 0,Y 338.054,Z 377.614,A -85,B 0,C 180,E1 -14463.374,E2 -14463.374} C_VEL
LIN {X 0,Y 336.677,Z 390.729,A -85,B 0,C 180,E1 -14465.893,E2 -14465.893} C_VEL
LIN {X 0,Y 338.402,Z 403.94,A -85,B 0,C 180,E1 -14466.359,E2 -14466.359} C_VEL
LIN {X 0,Y 341.874,Z 435.856,A -85,B 0,C 180,E1 -14467.311,E2 -14467.311} C_VEL
LIN {X 0,Y 342.849,Z 448.184,A -85,B 0,C 180,E1 -14467.648,E2 -14467.648} C_VEL
LIN {X 0,Y 341.836,Z 501.847,A -85,B 0,C 180,E1 -14468.795,E2 -14468.795} C_VEL
LIN {X 0,Y 341.031,Z 515.092,A -85,B 0,C 180,E1 -14469.295,E2 -14469.295} C_VEL
LIN {X 0,Y 340.023,Z 527.282,A -85,B 0,C 180,E1 -14469.981,E2 -14469.981} C_VEL
LIN {X 0,Y 338.651,Z 539.604,A -85,B 0,C 180,E1 -14470.922,E2 -14470.922} C_VEL
LIN {X 0,Y 337.177,Z 551.286,A -85,B 0,C 180,E1 -14472.095,E2 -14472.095} C_VEL
LIN {X 0,Y 335.727,Z 561.833,A -85,B 0,C 180,E1 -14473.428,E2 -14473.428} C_VEL
LIN {X 0,Y 334.694,Z 570.878,A -85,B 0,C 180,E1 -14474.845,E2 -14474.845} C_VEL
LIN {X 0,Y 333.73,Z 579.977,A -85,B 0,C 180,E1 -14476.606,E2 -14476.606} C_VEL
LIN {X 0,Y 333.016,Z 587.608,A -85,B 0,C 180,E1 -14478.435,E2 -14478.435} C_VEL
LIN {X 0,Y 332.65,Z 593.779,A -85,B 0,C 180,E1 -14480.269,E2 -14480.269} C_VEL
LIN {X 0,Y 332.577,Z 598.694,A -85,B 0,C 180,E1 -14482.105,E2 -14482.105} C_VEL
LIN {X 0,Y 332.75,Z 602.485,A -85,B 0,C 180,E1 -14483.938,E2 -14483.938} C_VEL
LIN {X 0,Y 332.946,Z 604.455,A -85,B 0,C 180,E1 -14485.157,E2 -14485.157} C_VEL
LIN {X 0,Y 333.092,Z 605.934,A -85,B 0,C 180,E1 -14486.371,E2 -14486.371} C_VEL
LIN {X 0,Y 333.526,Z 607.668,A -85,B 0,C 180,E1 -14488.793,E2 -14488.793} C_VEL
LIN {X 0,Y 333.645,Z 607.908,A -85,B 0,C 180,E1 -14490,E2 -14490} C_VEL
LIN {X 0,Y 333.526,Z 607.663,A -85,B 0,C 180,E1 -14491.207,E2 -14491.207} C_VEL
LIN {X 0,Y 333.098,Z 605.925,A -85,B 0,C 180,E1 -14493.629,E2 -14493.629} C_VEL
LIN {X 0,Y 332.958,Z 604.441,A -85,B 0,C 180,E1 -14494.843,E2 -14494.843} C_VEL
LIN {X 0,Y 332.719,Z 600.89,A -85,B 0,C 180,E1 -14496.89,E2 -14496.89} C_VEL
LIN {X 0,Y 332.584,Z 595.499,A -85,B 0,C 180,E1 -14499.119,E2 -14499.119} C_VEL
LIN {X 0,Y 332.825,Z 589.762,A -85,B 0,C 180,E1 -14500.955,E2 -14500.955} C_VEL
LIN {X 0,Y 333.363,Z 582.648,A -85,B 0,C 180,E1 -14502.789,E2 -14502.789} C_VEL
LIN {X 0,Y 334.131,Z 575.432,A -85,B 0,C 180,E1 -14504.308,E2 -14504.308} C_VEL
LIN {X 0,Y 335.206,Z 566.775,A -85,B 0,C 180,E1 -14505.816,E2 -14505.816} C_VEL
LIN {X 0,Y 336.324,Z 557.302,A -85,B 0,C 180,E1 -14507.167,E2 -14507.167} C_VEL
LIN {X 0,Y 337.831,Z 545.621,A -85,B 0,C 180,E1 -14508.496,E2 -14508.496} C_VEL
LIN {X 0,Y 339.275,Z 534.156,A -85,B 0,C 180,E1 -14509.513,E2 -14509.513} C_VEL
LIN {X 0,Y 340.439,Z 522.37,A -85,B 0,C 180,E1 -14510.308,E2 -14510.308} C_VEL
LIN {X 0,Y 341.386,Z 509.731,A -85,B 0,C 180,E1 -14510.919,E2 -14510.919} C_VEL
LIN {X 0,Y 341.921,Z 496.87,A -85,B 0,C 180,E1 -14511.318,E2 -14511.318} C_VEL
LIN {X 0,Y 342.824,Z 446.697,A -85,B 0,C 180,E1 -14512.369,E2 -14512.369} C_VEL
LIN {X 0,Y 339.619,Z 414.452,A -85,B 0,C 180,E1 -14513.3,E2 -14513.3} C_VEL
LIN {X 0,Y 336.651,Z 390.892,A -85,B 0,C 180,E1 -14514.071,E2 -14514.071} C_VEL
LIN {X 0,Y 338.984,Z 369.634,A -85,B 0,C 180,E1 -14518.142,E2 -14518.142} C_VEL
LIN {X 0,Y 340.116,Z 359.661,A -85,B 0,C 180,E1 -14520.072,E2 -14520.072} C_VEL
LIN {X 0,Y 339.839,Z 356.241,A -85,B 0,C 180,E1 -14520.786,E2 -14520.786} C_VEL
LIN {X 0,Y 336.894,Z 342.755,A -85,B 0,C 180,E1 -14523.79,E2 -14523.79} C_VEL
LIN {X 0,Y 333.686,Z 330.058,A -85,B 0,C 180,E1 -14526.837,E2 -14526.837} C_VEL
LIN {X 0,Y 333.6,Z 329.918,A -85,B 0,C 180,E1 -14530.773,E2 -14530.773} C_VEL
LIN {X 0,Y 333.585,Z 329.9,A -85,B 0,C 180,E1 -14534.249,E2 -14534.249} C_VEL
LIN {X 0,Y 333.633,Z 329.923,A -85,B 0,C 180,E1 -14537.617,E2 -14537.617} C_VEL
LIN {X 0,Y 333.611,Z 329.888,A -85,B 0,C 180,E1 -14541.21,E2 -14541.21} C_VEL
LIN {X 0,Y 333.668,Z 329.866,A -85,B 0,C 180,E1 -14543.86,E2 -14543.86} C_VEL
LIN {X 0,Y 333.639,Z 329.922,A -85,B 0,C 180,E1 -14547.413,E2 -14547.413} C_VEL
LIN {X 0,Y 333.648,Z 329.905,A -85,B 0,C 180,E1 -14551.022,E2 -14551.022} C_VEL
LIN {X 0,Y 333.661,Z 329.922,A -85,B 0,C 180,E1 -14555.085,E2 -14555.085} C_VEL
LIN {X 0,Y 333.66,Z 329.893,A -85,B 0,C 180,E1 -14559.018,E2 -14559.018} C_VEL
LIN {X 0,Y 333.788,Z 329.895,A -85,B 0,C 180,E1 -14561.589,E2 -14561.589} C_VEL
LIN {X 0,Y 333.803,Z 329.898,A -85,B 0,C 180,E1 -14565.576,E2 -14565.576} C_VEL
LIN {X 0,Y 333.81,Z 329.899,A -85,B 0,C 180,E1 -14569.077,E2 -14569.077} C_VEL
LIN {X 0,Y 333.965,Z 329.875,A -85,B 0,C 180,E1 -14572.746,E2 -14572.746} C_VEL
LIN {X 0,Y 333.775,Z 329.898,A -85,B 0,C 180,E1 -14575.169,E2 -14575.169} C_VEL
LIN {X 0,Y 334.058,Z 329.876,A -85,B 0,C 180,E1 -14577.589,E2 -14577.589} C_VEL
LIN {X 0,Y 334.052,Z 329.856,A -85,B 0,C 180,E1 -14581.206,E2 -14581.206} C_VEL
LIN {X 0,Y 334.063,Z 329.866,A -85,B 0,C 180,E1 -14582.412,E2 -14582.412} C_VEL
LIN {X 0,Y 333.949,Z 329.874,A -85,B 0,C 180,E1 -14586.523,E2 -14586.523} C_VEL
LIN {X 0,Y 333.814,Z 329.897,A -85,B 0,C 180,E1 -14589.697,E2 -14589.697} C_VEL
LIN {X 0,Y 333.787,Z 329.896,A -85,B 0,C 180,E1 -14593.392,E2 -14593.392} C_VEL
LIN {X 0,Y 333.713,Z 329.913,A -85,B 0,C 180,E1 -14597.148,E2 -14597.148} C_VEL
LIN {X 0,Y 333.682,Z 329.911,A -85,B 0,C 180,E1 -14599.694,E2 -14599.694} C_VEL
LIN {X 0,Y 333.637,Z 329.927,A -85,B 0,C 180,E1 -14603.593,E2 -14603.593} C_VEL
LIN {X 0,Y 333.623,Z 329.916,A -85,B 0,C 180,E1 -14606.256,E2 -14606.256} C_VEL
LIN {X 0,Y 333.623,Z 329.881,A -85,B 0,C 180,E1 -14608.981,E2 -14608.981} C_VEL
LIN {X 0,Y 333.638,Z 329.914,A -85,B 0,C 180,E1 -14612.587,E2 -14612.587} C_VEL
LIN {X 0,Y 333.671,Z 329.915,A -85,B 0,C 180,E1 -14616.14,E2 -14616.14} C_VEL
LIN {X 0,Y 333.598,Z 329.895,A -85,B 0,C 180,E1 -14619.199,E2 -14619.199} C_VEL
LIN {X 0,Y 333.623,Z 329.925,A -85,B 0,C 180,E1 -14622.499,E2 -14622.499} C_VEL
LIN {X 0,Y 333.59,Z 329.91,A -85,B 0,C 180,E1 -14625.955,E2 -14625.955} C_VEL
LIN {X 0,Y 333.599,Z 329.928,A -85,B 0,C 180,E1 -14629.325,E2 -14629.325} C_VEL
LIN {X 0,Y 333.66,Z 329.905,A -85,B 0,C 180,E1 -14633.17,E2 -14633.17} C_VEL
LIN {X 0,Y 333.671,Z 329.924,A -85,B 0,C 180,E1 -14635.342,E2 -14635.342} C_VEL
LIN {X 0,Y 333.628,Z 329.918,A -85,B 0,C 180,E1 -14638.222,E2 -14638.222} C_VEL
LIN {X 0,Y 333.629,Z 329.903,A -85,B 0,C 180,E1 -14641.021,E2 -14641.021} C_VEL
LIN {X 0,Y 333.694,Z 329.915,A -85,B 0,C 180,E1 -14645.089,E2 -14645.089} C_VEL
LIN {X 0,Y 333.718,Z 330.116,A -85,B 0,C 180,E1 -14646.167,E2 -14646.167} C_VEL
LIN {X 0,Y 333.994,Z 331.249,A -85,B 0,C 180,E1 -14646.38,E2 -14646.38} C_VEL
LIN {X 0,Y 343.877,Z 353.339,A -85,B 0,C 180,E1 -14647.639,E2 -14647.639} C_VEL
LIN {X 0,Y 344.507,Z 355.329,A -85,B 0,C 180,E1 -14647.728,E2 -14647.728} C_VEL
LIN {X 0,Y 343.743,Z 407.327,A -85,B 0,C 180,E1 -14648.83,E2 -14648.83} C_VEL
LIN {X 0,Y 343.597,Z 419.934,A -85,B 0,C 180,E1 -14649.237,E2 -14649.237} C_VEL
LIN {X 0,Y 343.148,Z 432.363,A -85,B 0,C 180,E1 -14649.859,E2 -14649.859} C_VEL
LIN {X 0,Y 342.488,Z 444.697,A -85,B 0,C 180,E1 -14650.725,E2 -14650.725} C_VEL
LIN {X 0,Y 341.524,Z 456.19,A -85,B 0,C 180,E1 -14651.788,E2 -14651.788} C_VEL
LIN {X 0,Y 340.383,Z 466.941,A -85,B 0,C 180,E1 -14653.044,E2 -14653.044} C_VEL
LIN {X 0,Y 339.311,Z 476.143,A -85,B 0,C 180,E1 -14654.38,E2 -14654.38} C_VEL
LIN {X 0,Y 338.352,Z 484.501,A -85,B 0,C 180,E1 -14655.874,E2 -14655.874} C_VEL
LIN {X 0,Y 337.202,Z 492.623,A -85,B 0,C 180,E1 -14657.665,E2 -14657.665} C_VEL
LIN {X 0,Y 336.138,Z 499.734,A -85,B 0,C 180,E1 -14659.638,E2 -14659.638} C_VEL
LIN {X 0,Y 335.461,Z 505.11,A -85,B 0,C 180,E1 -14661.567,E2 -14661.567} C_VEL
LIN {X 0,Y 334.721,Z 509.004,A -85,B 0,C 180,E1 -14663.369,E2 -14663.369} C_VEL
LIN {X 0,Y 334.172,Z 511.877,A -85,B 0,C 180,E1 -14665.174,E2 -14665.174} C_VEL
LIN {X 0,Y 334.141,Z 513.221,A -85,B 0,C 180,E1 -14666.382,E2 -14666.382} C_VEL
LIN {X 0,Y 333.939,Z 514.201,A -85,B 0,C 180,E1 -14667.588,E2 -14667.588} C_VEL
LIN {X 0,Y 333.984,Z 514.781,A -85,B 0,C 180,E1 -14668.794,E2 -14668.794} C_VEL
LIN {X 0,Y 333.961,Z 515.008,A -85,B 0,C 180,E1 -14670,E2 -14670} C_VEL
LIN {X 0,Y 333.984,Z 514.822,A -85,B 0,C 180,E1 -14671.206,E2 -14671.206} C_VEL
LIN {X 0,Y 333.938,Z 514.268,A -85,B 0,C 180,E1 -14672.412,E2 -14672.412} C_VEL
LIN {X 0,Y 334.137,Z 513.315,A -85,B 0,C 180,E1 -14673.618,E2 -14673.618} C_VEL
LIN {X 0,Y 334.161,Z 512.014,A -85,B 0,C 180,E1 -14674.826,E2 -14674.826} C_VEL
LIN {X 0,Y 334.716,Z 509.191,A -85,B 0,C 180,E1 -14676.631,E2 -14676.631} C_VEL
LIN {X 0,Y 335.436,Z 505.363,A -85,B 0,C 180,E1 -14678.433,E2 -14678.433} C_VEL
LIN {X 0,Y 336.072,Z 500.284,A -85,B 0,C 180,E1 -14680.299,E2 -14680.299} C_VEL
LIN {X 0,Y 337.213,Z 493.044,A -85,B 0,C 180,E1 -14682.335,E2 -14682.335} C_VEL
LIN {X 0,Y 338.342,Z 485.015,A -85,B 0,C 180,E1 -14684.127,E2 -14684.127} C_VEL
LIN {X 0,Y 339.32,Z 476.792,A -85,B 0,C 180,E1 -14685.62,E2 -14685.62} C_VEL
LIN {X 0,Y 340.332,Z 467.756,A -85,B 0,C 180,E1 -14686.959,E2 -14686.959} C_VEL
LIN {X 0,Y 341.517,Z 457.243,A -85,B 0,C 180,E1 -14688.204,E2 -14688.204} C_VEL
LIN {X 0,Y 342.46,Z 445.571,A -85,B 0,C 180,E1 -14689.308,E2 -14689.308} C_VEL
LIN {X 0,Y 343.219,Z 434.12,A -85,B 0,C 180,E1 -14690.136,E2 -14690.136} C_VEL
LIN {X 0,Y 343.634,Z 421.619,A -85,B 0,C 180,E1 -14690.798,E2 -14690.798} C_VEL
LIN {X 0,Y 343.736,Z 411.57,A -85,B 0,C 180,E1 -14691.169,E2 -14691.169} C_VEL
LIN {X 0,Y 344.168,Z 373.082,A -85,B 0,C 180,E1 -14692.012,E2 -14692.012} C_VEL
LIN {X 0,Y 344.51,Z 354.843,A -85,B 0,C 180,E1 -14692.392,E2 -14692.392} C_VEL
LIN {X 0,Y 334.655,Z 332.683,A -85,B 0,C 180,E1 -14693.634,E2 -14693.634} C_VEL
LIN {X 0,Y 333.779,Z 330.458,A -85,B 0,C 180,E1 -14693.829,E2 -14693.829} C_VEL
LIN {X 0,Y 333.689,Z 329.939,A -85,B 0,C 180,E1 -14694.083,E2 -14694.083} C_VEL
LIN {X 0,Y 333.642,Z 329.884,A -85,B 0,C 180,E1 -14697.784,E2 -14697.784} C_VEL
LIN {X 0,Y 333.655,Z 329.923,A -85,B 0,C 180,E1 -14700.366,E2 -14700.366} C_VEL
LIN {X 0,Y 333.631,Z 329.914,A -85,B 0,C 180,E1 -14702.385,E2 -14702.385} C_VEL
LIN {X 0,Y 333.005,Z 329.996,A -85,B 0,C 180,E1 -14703.392,E2 -14703.392} C_VEL
LIN {X 0,Y 330.182,Z 330.357,A -85,B 0,C 180,E1 -14705.031,E2 -14705.031} C_VEL
LIN {X 0,Y 327.75,Z 330.648,A -85,B 0,C 180,E1 -14706.359,E2 -14706.359} C_VEL
LIN {X 0,Y 326.678,Z 330.773,A -85,B 0,C 180,E1 -14707.387,E2 -14707.387} C_VEL
LIN {X 0,Y 326.578,Z 330.786,A -85,B 0,C 180,E1 -14707.735,E2 -14707.735} C_VEL
LIN {X 0,Y 326.541,Z 330.804,A -85,B 0,C 180,E1 -14711.123,E2 -14711.123} C_VEL
LIN {X 0,Y 326.556,Z 330.782,A -85,B 0,C 180,E1 -14713.526,E2 -14713.526} C_VEL
LIN {X 0,Y 326.568,Z 330.807,A -85,B 0,C 180,E1 -14717.028,E2 -14717.028} C_VEL
LIN {X 0,Y 326.567,Z 330.77,A -85,B 0,C 180,E1 -14720.781,E2 -14720.781} C_VEL
LIN {X 0,Y 326.608,Z 330.799,A -85,B 0,C 180,E1 -14724.48,E2 -14724.48} C_VEL
LIN {X 0,Y 326.603,Z 330.79,A -85,B 0,C 180,E1 -14727.455,E2 -14727.455} C_VEL
LIN {X 0,Y 326.574,Z 330.755,A -85,B 0,C 180,E1 -14730.332,E2 -14730.332} C_VEL
LIN {X 0,Y 326.59,Z 330.783,A -85,B 0,C 180,E1 -14733.134,E2 -14733.134} C_VEL
LIN {X 0,Y 326.586,Z 330.799,A -85,B 0,C 180,E1 -14737.21,E2 -14737.21} C_VEL
LIN {X 0,Y 326.666,Z 330.792,A -85,B 0,C 180,E1 -14741.193,E2 -14741.193} C_VEL
LIN {X 0,Y 326.758,Z 330.763,A -85,B 0,C 180,E1 -14745.433,E2 -14745.433} C_VEL
LIN {X 0,Y 326.75,Z 330.783,A -85,B 0,C 180,E1 -14748.838,E2 -14748.838} C_VEL
LIN {X 0,Y 326.904,Z 330.749,A -85,B 0,C 180,E1 -14752.589,E2 -14752.589} C_VEL
LIN {X 0,Y 326.744,Z 330.783,A -85,B 0,C 180,E1 -14755.064,E2 -14755.064} C_VEL
LIN {X 0,Y 327.006,Z 330.745,A -85,B 0,C 180,E1 -14757.536,E2 -14757.536} C_VEL
LIN {X 0,Y 327.038,Z 330.742,A -85,B 0,C 180,E1 -14761.231,E2 -14761.231} C_VEL
LIN {X 0,Y 326.744,Z 330.782,A -85,B 0,C 180,E1 -14763.7,E2 -14763.7} C_VEL
LIN {X 0,Y 326.944,Z 330.742,A -85,B 0,C 180,E1 -14766.17,E2 -14766.17} C_VEL
LIN {X 0,Y 326.775,Z 330.78,A -85,B 0,C 180,E1 -14769.907,E2 -14769.907} C_VEL
LIN {X 0,Y 326.753,Z 330.769,A -85,B 0,C 180,E1 -14773.686,E2 -14773.686} C_VEL
LIN {X 0,Y 326.659,Z 330.792,A -85,B 0,C 180,E1 -14777.53,E2 -14777.53} C_VEL
LIN {X 0,Y 326.625,Z 330.769,A -85,B 0,C 180,E1 -14780.137,E2 -14780.137} C_VEL
LIN {X 0,Y 326.607,Z 330.801,A -85,B 0,C 180,E1 -14784.132,E2 -14784.132} C_VEL
LIN {X 0,Y 326.594,Z 330.782,A -85,B 0,C 180,E1 -14788.257,E2 -14788.257} C_VEL
LIN {X 0,Y 326.569,Z 330.805,A -85,B 0,C 180,E1 -14791.098,E2 -14791.098} C_VEL
LIN {X 0,Y 326.602,Z 330.788,A -85,B 0,C 180,E1 -14794.02,E2 -14794.02} C_VEL
LIN {X 0,Y 326.617,Z 330.8,A -85,B 0,C 180,E1 -14797.237,E2 -14797.237} C_VEL
LIN {X 0,Y 326.54,Z 330.809,A -85,B 0,C 180,E1 -14801.125,E2 -14801.125} C_VEL
LIN {X 0,Y 326.555,Z 330.783,A -85,B 0,C 180,E1 -14803.527,E2 -14803.527} C_VEL
LIN {X 0,Y 326.568,Z 330.795,A -85,B 0,C 180,E1 -14807.03,E2 -14807.03} C_VEL
LIN {X 0,Y 326.568,Z 330.784,A -85,B 0,C 180,E1 -14810.782,E2 -14810.782} C_VEL
LIN {X 0,Y 326.626,Z 331.041,A -85,B 0,C 180,E1 -14812.67,E2 -14812.67} C_VEL
LIN {X 0,Y 329.633,Z 342.809,A -85,B 0,C 180,E1 -14815.574,E2 -14815.574} C_VEL
LIN {X 0,Y 332.471,Z 355.268,A -85,B 0,C 180,E1 -14818.455,E2 -14818.455} C_VEL
LIN {X 0,Y 333.291,Z 360.479,A -85,B 0,C 180,E1 -14819.598,E2 -14819.598} C_VEL
LIN {X 0,Y 331.505,Z 375.075,A -85,B 0,C 180,E1 -14822.485,E2 -14822.485} C_VEL
LIN {X 0,Y 329.875,Z 389.834,A -85,B 0,C 180,E1 -14825.377,E2 -14825.377} C_VEL
LIN {X 0,Y 333.386,Z 417.817,A -85,B 0,C 180,E1 -14826.316,E2 -14826.316} C_VEL
LIN {X 0,Y 336.261,Z 447.158,A -85,B 0,C 180,E1 -14827.184,E2 -14827.184} C_VEL
LIN {X 0,Y 335.172,Z 500.865,A -85,B 0,C 180,E1 -14828.352,E2 -14828.352} C_VEL
LIN {X 0,Y 334.423,Z 514.116,A -85,B 0,C 180,E1 -14828.867,E2 -14828.867} C_VEL
LIN {X 0,Y 333.243,Z 527.424,A -85,B 0,C 180,E1 -14829.637,E2 -14829.637} C_VEL
LIN {X 0,Y 331.915,Z 538.615,A -85,B 0,C 180,E1 -14830.52,E2 -14830.52} C_VEL
LIN {X 0,Y 330.409,Z 550.299,A -85,B 0,C 180,E1 -14831.715,E2 -14831.715} C_VEL
LIN {X 0,Y 328.938,Z 560.849,A -85,B 0,C 180,E1 -14833.076,E2 -14833.076} C_VEL
LIN {X 0,Y 327.839,Z 569.528,A -85,B 0,C 180,E1 -14834.458,E2 -14834.458} C_VEL
LIN {X 0,Y 327.052,Z 576.21,A -85,B 0,C 180,E1 -14835.728,E2 -14835.728} C_VEL
LIN {X 0,Y 326.185,Z 584.26,A -85,B 0,C 180,E1 -14837.558,E2 -14837.558} C_VEL
LIN {X 0,Y 325.677,Z 590.895,A -85,B 0,C 180,E1 -14839.431,E2 -14839.431} C_VEL
LIN {X 0,Y 325.486,Z 596.203,A -85,B 0,C 180,E1 -14841.307,E2 -14841.307} C_VEL
LIN {X 0,Y 325.62,Z 600.289,A -85,B 0,C 180,E1 -14843.14,E2 -14843.14} C_VEL
LIN {X 0,Y 325.866,Z 603.467,A -85,B 0,C 180,E1 -14845.051,E2 -14845.051} C_VEL
LIN {X 0,Y 326.043,Z 604.951,A -85,B 0,C 180,E1 -14846.292,E2 -14846.292} C_VEL
LIN {X 0,Y 326.465,Z 606.686,A -85,B 0,C 180,E1 -14848.766,E2 -14848.766} C_VEL
LIN {X 0,Y 326.617,Z 606.93,A -85,B 0,C 180,E1 -14850,E2 -14850} C_VEL
LIN {X 0,Y 326.465,Z 606.68,A -85,B 0,C 180,E1 -14851.233,E2 -14851.233} C_VEL
LIN {X 0,Y 326.049,Z 604.941,A -85,B 0,C 180,E1 -14853.708,E2 -14853.708} C_VEL
LIN {X 0,Y 325.878,Z 603.452,A -85,B 0,C 180,E1 -14854.949,E2 -14854.949} C_VEL
LIN {X 0,Y 325.652,Z 600.174,A -85,B 0,C 180,E1 -14856.906,E2 -14856.906} C_VEL
LIN {X 0,Y 325.49,Z 596.165,A -85,B 0,C 180,E1 -14858.693,E2 -14858.693} C_VEL
LIN {X 0,Y 325.726,Z 589.809,A -85,B 0,C 180,E1 -14860.882,E2 -14860.882} C_VEL
LIN {X 0,Y 326.274,Z 582.921,A -85,B 0,C 180,E1 -14862.755,E2 -14862.755} C_VEL
LIN {X 0,Y 327.091,Z 575.101,A -85,B 0,C 180,E1 -14864.483,E2 -14864.483} C_VEL
LIN {X 0,Y 328.318,Z 565.775,A -85,B 0,C 180,E1 -14866.157,E2 -14866.157} C_VEL
LIN {X 0,Y 329.347,Z 557.466,A -85,B 0,C 180,E1 -14867.382,E2 -14867.382} C_VEL
LIN {X 0,Y 330.887,Z 546.064,A -85,B 0,C 180,E1 -14868.738,E2 -14868.738} C_VEL
LIN {X 0,Y 332.335,Z 534.937,A -85,B 0,C 180,E1 -14869.776,E2 -14869.776} C_VEL
LIN {X 0,Y 333.66,Z 522.615,A -85,B 0,C 180,E1 -14870.659,E2 -14870.659} C_VEL
LIN {X 0,Y 334.676,Z 509.645,A -85,B 0,C 180,E1 -14871.318,E2 -14871.318} C_VEL
LIN {X 0,Y 335.29,Z 495.861,A -85,B 0,C 180,E1 -14871.761,E2 -14871.761} C_VEL
LIN {X 0,Y 336.194,Z 446.889,A -85,B 0,C 180,E1 -14872.807,E2 -14872.807} C_VEL
LIN {X 0,Y 332.851,Z 413.402,A -85,B 0,C 180,E1 -14873.803,E2 -14873.803} C_VEL
LIN {X 0,Y 329.873,Z 390.185,A -85,B 0,C 180,E1 -14874.574,E2 -14874.574} C_VEL
LIN {X 0,Y 330.232,Z 386.677,A -85,B 0,C 180,E1 -14875.191,E2 -14875.191} C_VEL
LIN {X 0,Y 332.689,Z 365.542,A -85,B 0,C 180,E1 -14879.371,E2 -14879.371} C_VEL
LIN {X 0,Y 333.254,Z 360.347,A -85,B 0,C 180,E1 -14880.406,E2 -14880.406} C_VEL
LIN {X 0,Y 331.695,Z 351.65,A -85,B 0,C 180,E1 -14882.343,E2 -14882.343} C_VEL
LIN {X 0,Y 328.79,Z 339.253,A -85,B 0,C 180,E1 -14885.248,E2 -14885.248} C_VEL
LIN {X 0,Y 326.606,Z 330.913,A -85,B 0,C 180,E1 -14887.356,E2 -14887.356} C_VEL
LIN {X 0,Y 326.54,Z 330.803,A -85,B 0,C 180,E1 -14891.124,E2 -14891.124} C_VEL
LIN {X 0,Y 326.555,Z 330.785,A -85,B 0,C 180,E1 -14893.526,E2 -14893.526} C_VEL
LIN {X 0,Y 326.568,Z 330.796,A -85,B 0,C 180,E1 -14897.028,E2 -14897.028} C_VEL
LIN {X 0,Y 326.567,Z 330.773,A -85,B 0,C 180,E1 -14900.781,E2 -14900.781} C_VEL
LIN {X 0,Y 326.62,Z 330.737,A -85,B 0,C 180,E1 -14902.952,E2 -14902.952} C_VEL
LIN {X 0,Y 326.602,Z 330.783,A -85,B 0,C 180,E1 -14905.98,E2 -14905.98} C_VEL
LIN {X 0,Y 326.607,Z 330.798,A -85,B 0,C 180,E1 -14909.397,E2 -14909.397} C_VEL
LIN {X 0,Y 326.598,Z 330.792,A -85,B 0,C 180,E1 -14913.135,E2 -14913.135} C_VEL
LIN {X 0,Y 326.607,Z 330.8,A -85,B 0,C 180,E1 -14915.868,E2 -14915.868} C_VEL
LIN {X 0,Y 326.649,Z 330.767,A -85,B 0,C 180,E1 -14919.864,E2 -14919.864} C_VEL
LIN {X 0,Y 326.694,Z 330.788,A -85,B 0,C 180,E1 -14922.472,E2 -14922.472} C_VEL
LIN {X 0,Y 326.753,Z 330.768,A -85,B 0,C 180,E1 -14926.314,E2 -14926.314} C_VEL
LIN {X 0,Y 326.777,Z 330.781,A -85,B 0,C 180,E1 -14930.093,E2 -14930.093} C_VEL
LIN {X 0,Y 326.946,Z 330.743,A -85,B 0,C 180,E1 -14933.83,E2 -14933.83} C_VEL
LIN {X 0,Y 327.002,Z 330.754,A -85,B 0,C 180,E1 -14937.536,E2 -14937.536} C_VEL
LIN {X 0,Y 327.022,Z 330.731,A -85,B 0,C 180,E1 -14941.231,E2 -14941.231} C_VEL
LIN {X 0,Y 326.755,Z 330.783,A -85,B 0,C 180,E1 -14943.7,E2 -14943.7} C_VEL
LIN {X 0,Y 326.911,Z 330.75,A -85,B 0,C 180,E1 -14946.512,E2 -14946.512} C_VEL
LIN {X 0,Y 326.777,Z 330.776,A -85,B 0,C 180,E1 -14949.907,E2 -14949.907} C_VEL
LIN {X 0,Y 326.751,Z 330.768,A -85,B 0,C 180,E1 -14953.686,E2 -14953.686} C_VEL
LIN {X 0,Y 326.658,Z 330.796,A -85,B 0,C 180,E1 -14957.53,E2 -14957.53} C_VEL
LIN {X 0,Y 326.625,Z 330.786,A -85,B 0,C 180,E1 -14960.138,E2 -14960.138} C_VEL
LIN {X 0,Y 326.586,Z 330.799,A -85,B 0,C 180,E1 -14962.79,E2 -14962.79} C_VEL
LIN {X 0,Y 326.59,Z 330.784,A -85,B 0,C 180,E1 -14966.866,E2 -14966.866} C_VEL
LIN {X 0,Y 326.566,Z 330.77,A -85,B 0,C 180,E1 -14971.098,E2 -14971.098} C_VEL
LIN {X 0,Y 326.603,Z 330.802,A -85,B 0,C 180,E1 -14974.02,E2 -14974.02} C_VEL
LIN {X 0,Y 326.619,Z 330.781,A -85,B 0,C 180,E1 -14977.238,E2 -14977.238} C_VEL
LIN {X 0,Y 326.539,Z 330.793,A -85,B 0,C 180,E1 -14981.125,E2 -14981.125} C_VEL
LIN {X 0,Y 326.556,Z 330.809,A -85,B 0,C 180,E1 -14983.527,E2 -14983.527} C_VEL
LIN {X 0,Y 326.569,Z 330.779,A -85,B 0,C 180,E1 -14987.03,E2 -14987.03} C_VEL
LIN {X 0,Y 326.579,Z 330.794,A -85,B 0,C 180,E1 -14991.386,E2 -14991.386} C_VEL
LIN {X 0,Y 326.616,Z 330.799,A -85,B 0,C 180,E1 -14994.853,E2 -14994.853} C_VEL
LIN {X 0,Y 326.607,Z 330.788,A -85,B 0,C 180,E1 -14997.456,E2 -14997.456} C_VEL
LIN {X 0,Y 326.58,Z 330.795,A -85,B 0,C 180,E1 -15000.333,E2 -15000.333} C_VEL
LIN {X 0,Y 326.605,Z 330.761,A -85,B 0,C 180,E1 -15003.136,E2 -15003.136} C_VEL
LIN {X 0,Y 326.687,Z 331.007,A -85,B 0,C 180,E1 -15005.621,E2 -15005.621} C_VEL
LIN {X 0,Y 326.966,Z 332.091,A -85,B 0,C 180,E1 -15005.833,E2 -15005.833} C_VEL
LIN {X 0,Y 337.171,Z 354.683,A -85,B 0,C 180,E1 -15007.176,E2 -15007.176} C_VEL
LIN {X 0,Y 337.965,Z 356.688,A -85,B 0,C 180,E1 -15007.281,E2 -15007.281} C_VEL
LIN {X 0,Y 337.193,Z 407.582,A -85,B 0,C 180,E1 -15008.379,E2 -15008.379} C_VEL
LIN {X 0,Y 337.077,Z 419.526,A -85,B 0,C 180,E1 -15008.754,E2 -15008.754} C_VEL
LIN {X 0,Y 336.585,Z 432.068,A -85,B 0,C 180,E1 -15009.369,E2 -15009.369} C_VEL
LIN {X 0,Y 335.931,Z 444.651,A -85,B 0,C 180,E1 -15010.246,E2 -15010.246} C_VEL
LIN {X 0,Y 334.997,Z 456.114,A -85,B 0,C 180,E1 -15011.301,E2 -15011.301} C_VEL
LIN {X 0,Y 333.959,Z 465.611,A -85,B 0,C 180,E1 -15012.392,E2 -15012.392} C_VEL
LIN {X 0,Y 333.021,Z 473.279,A -85,B 0,C 180,E1 -15013.447,E2 -15013.447} C_VEL
LIN {X 0,Y 331.937,Z 482.318,A -85,B 0,C 180,E1 -15014.968,E2 -15014.968} C_VEL
LIN {X 0,Y 330.688,Z 491.09,A -85,B 0,C 180,E1 -15016.793,E2 -15016.793} C_VEL
LIN {X 0,Y 329.778,Z 497.266,A -85,B 0,C 180,E1 -15018.382,E2 -15018.382} C_VEL
LIN {X 0,Y 328.961,Z 502.877,A -85,B 0,C 180,E1 -15020.159,E2 -15020.159} C_VEL
LIN {X 0,Y 328.184,Z 507.491,A -85,B 0,C 180,E1 -15021.999,E2 -15021.999} C_VEL
LIN {X 0,Y 327.49,Z 511.032,A -85,B 0,C 180,E1 -15023.84,E2 -15023.84} C_VEL
LIN {X 0,Y 327.166,Z 512.856,A -85,B 0,C 180,E1 -15025.071,E2 -15025.071} C_VEL
LIN {X 0,Y 327.126,Z 514.2,A -85,B 0,C 180,E1 -15026.305,E2 -15026.305} C_VEL
LIN {X 0,Y 326.917,Z 515.179,A -85,B 0,C 180,E1 -15027.536,E2 -15027.536} C_VEL
LIN {X 0,Y 326.958,Z 515.759,A -85,B 0,C 180,E1 -15028.768,E2 -15028.768} C_VEL
LIN {X 0,Y 326.934,Z 515.985,A -85,B 0,C 180,E1 -15030,E2 -15030} C_VEL
LIN {X 0,Y 326.958,Z 515.799,A -85,B 0,C 180,E1 -15031.232,E2 -15031.232} C_VEL
LIN {X 0,Y 326.917,Z 515.245,A -85,B 0,C 180,E1 -15032.464,E2 -15032.464} C_VEL
LIN {X 0,Y 327.122,Z 514.293,A -85,B 0,C 180,E1 -15033.695,E2 -15033.695} C_VEL
LIN {X 0,Y 327.154,Z 512.992,A -85,B 0,C 180,E1 -15034.929,E2 -15034.929} C_VEL
LIN {X 0,Y 327.737,Z 510.168,A -85,B 0,C 180,E1 -15036.773,E2 -15036.773} C_VEL
LIN {X 0,Y 328.486,Z 506.34,A -85,B 0,C 180,E1 -15038.613,E2 -15038.613} C_VEL
LIN {X 0,Y 329.159,Z 501.26,A -85,B 0,C 180,E1 -15040.518,E2 -15040.518} C_VEL
LIN {X 0,Y 330.351,Z 494.019,A -85,B 0,C 180,E1 -15042.595,E2 -15042.595} C_VEL
LIN {X 0,Y 331.53,Z 485.991,A -85,B 0,C 180,E1 -15044.423,E2 -15044.423} C_VEL
LIN {X 0,Y 332.554,Z 477.767,A -85,B 0,C 180,E1 -15045.946,E2 -15045.946} C_VEL
LIN {X 0,Y 333.614,Z 468.731,A -85,B 0,C 180,E1 -15047.311,E2 -15047.311} C_VEL
LIN {X 0,Y 334.85,Z 458.216,A -85,B 0,C 180,E1 -15048.58,E2 -15048.58} C_VEL
LIN {X 0,Y 335.836,Z 446.543,A -85,B 0,C 180,E1 -15049.705,E2 -15049.705} C_VEL
LIN {X 0,Y 336.626,Z 435.09,A -85,B 0,C 180,E1 -15050.548,E2 -15050.548} C_VEL
LIN {X 0,Y 337.065,Z 422.758,A -85,B 0,C 180,E1 -15051.215,E2 -15051.215} C_VEL
LIN {X 0,Y 337.157,Z 413.021,A -85,B 0,C 180,E1 -15051.589,E2 -15051.589} C_VEL
LIN {X 0,Y 337.577,Z 375.231,A -85,B 0,C 180,E1 -15052.438,E2 -15052.438} C_VEL
LIN {X 0,Y 337.967,Z 356.65,A -85,B 0,C 180,E1 -15052.831,E2 -15052.831} C_VEL
LIN {X 0,Y 329.041,Z 336.489,A -85,B 0,C 180,E1 -15053.992,E2 -15053.992} C_VEL
LIN {X 0,Y 326.83,Z 331.602,A -85,B 0,C 180,E1 -15054.33,E2 -15054.33} C_VEL
LIN {X 0,Y 326.679,Z 330.83,A -85,B 0,C 180,E1 -15054.588,E2 -15054.588} C_VEL
LIN {X 0,Y 326.589,Z 330.765,A -85,B 0,C 180,E1 -15058.256,E2 -15058.256} C_VEL
LIN {X 0,Y 326.571,Z 330.805,A -85,B 0,C 180,E1 -15061.097,E2 -15061.097} C_VEL
LIN {X 0,Y 326.605,Z 330.799,A -85,B 0,C 180,E1 -15064.019,E2 -15064.019} C_VEL
LIN {X 0,Y 326.578,Z 330.786,A -85,B 0,C 180,E1 -15067.735,E2 -15067.735} C_VEL
LIN {X 0,Y 325.889,Z 330.882,A -85,B 0,C 180,E1 -15068.764,E2 -15068.764} C_VEL
LIN {X 0,Y 323.071,Z 331.244,A -85,B 0,C 180,E1 -15070.441,E2 -15070.441} C_VEL
LIN {X 0,Y 320.683,Z 331.526,A -85,B 0,C 180,E1 -15071.799,E2 -15071.799} C_VEL
LIN {X 0,Y 319.631,Z 331.644,A -85,B 0,C 180,E1 -15072.849,E2 -15072.849} C_VEL
LIN {X 0,Y 319.53,Z 331.656,A -85,B 0,C 180,E1 -15073.205,E2 -15073.205} C_VEL
LIN {X 0,Y 319.547,Z 331.682,A -85,B 0,C 180,E1 -15077.015,E2 -15077.015} C_VEL
LIN {X 0,Y 319.511,Z 331.65,A -85,B 0,C 180,E1 -15080.365,E2 -15080.365} C_VEL
LIN {X 0,Y 319.576,Z 331.675,A -85,B 0,C 180,E1 -15084.457,E2 -15084.457} C_VEL
LIN {X 0,Y 319.518,Z 331.659,A -85,B 0,C 180,E1 -15088.136,E2 -15088.136} C_VEL
LIN {X 0,Y 319.538,Z 331.638,A -85,B 0,C 180,E1 -15091.613,E2 -15091.613} C_VEL
LIN {X 0,Y 319.521,Z 331.682,A -85,B 0,C 180,E1 -15095.297,E2 -15095.297} C_VEL
LIN {X 0,Y 319.558,Z 331.671,A -85,B 0,C 180,E1 -15098.045,E2 -15098.045} C_VEL
LIN {X 0,Y 319.608,Z 331.673,A -85,B 0,C 180,E1 -15102.07,E2 -15102.07} C_VEL
LIN {X 0,Y 319.725,Z 331.641,A -85,B 0,C 180,E1 -15106.007,E2 -15106.007} C_VEL
LIN {X 0,Y 319.729,Z 331.657,A -85,B 0,C 180,E1 -15109.872,E2 -15109.872} C_VEL
LIN {X 0,Y 319.889,Z 331.629,A -85,B 0,C 180,E1 -15113.693,E2 -15113.693} C_VEL
LIN {X 0,Y 319.953,Z 331.624,A -85,B 0,C 180,E1 -15117.482,E2 -15117.482} C_VEL
LIN {X 0,Y 320.006,Z 331.618,A -85,B 0,C 180,E1 -15121.258,E2 -15121.258} C_VEL
LIN {X 0,Y 319.713,Z 331.647,A -85,B 0,C 180,E1 -15125.044,E2 -15125.044} C_VEL
LIN {X 0,Y 319.853,Z 331.633,A -85,B 0,C 180,E1 -15127.576,E2 -15127.576} C_VEL
LIN {X 0,Y 319.706,Z 331.654,A -85,B 0,C 180,E1 -15131.411,E2 -15131.411} C_VEL
LIN {X 0,Y 319.708,Z 331.658,A -85,B 0,C 180,E1 -15134.712,E2 -15134.712} C_VEL
LIN {X 0,Y 319.635,Z 331.652,A -85,B 0,C 180,E1 -15139.012,E2 -15139.012} C_VEL
LIN {X 0,Y 319.537,Z 331.676,A -85,B 0,C 180,E1 -15143.322,E2 -15143.322} C_VEL
LIN {X 0,Y 319.548,Z 331.676,A -85,B 0,C 180,E1 -15146.096,E2 -15146.096} C_VEL
LIN {X 0,Y 319.538,Z 331.662,A -85,B 0,C 180,E1 -15148.939,E2 -15148.939} C_VEL
LIN {X 0,Y 319.52,Z 331.686,A -85,B 0,C 180,E1 -15151.863,E2 -15151.863} C_VEL
LIN {X 0,Y 319.573,Z 331.667,A -85,B 0,C 180,E1 -15155.543,E2 -15155.543} C_VEL
LIN {X 0,Y 319.525,Z 331.671,A -85,B 0,C 180,E1 -15159.663,E2 -15159.663} C_VEL
LIN {X 0,Y 319.515,Z 331.66,A -85,B 0,C 180,E1 -15163.46,E2 -15163.46} C_VEL
LIN {X 0,Y 319.547,Z 331.668,A -85,B 0,C 180,E1 -15167.016,E2 -15167.016} C_VEL
LIN {X 0,Y 319.512,Z 331.661,A -85,B 0,C 180,E1 -15170.367,E2 -15170.367} C_VEL
LIN {X 0,Y 319.57,Z 331.914,A -85,B 0,C 180,E1 -15172.139,E2 -15172.139} C_VEL
LIN {X 0,Y 322.63,Z 343.621,A -85,B 0,C 180,E1 -15175.124,E2 -15175.124} C_VEL
LIN {X 0,Y 325.436,Z 356.103,A -85,B 0,C 180,E1 -15178.091,E2 -15178.091} C_VEL
LIN {X 0,Y 326.41,Z 362.158,A -85,B 0,C 180,E1 -15179.457,E2 -15179.457} C_VEL
LIN {X 0,Y 324.216,Z 379.264,A -85,B 0,C 180,E1 -15182.922,E2 -15182.922} C_VEL
LIN {X 0,Y 323.145,Z 388.643,A -85,B 0,C 180,E1 -15184.808,E2 -15184.808} C_VEL
LIN {X 0,Y 324.121,Z 396.501,A -85,B 0,C 180,E1 -15185.123,E2 -15185.123} C_VEL
LIN {X 0,Y 328.31,Z 432.234,A -85,B 0,C 180,E1 -15186.28,E2 -15186.28} C_VEL
LIN {X 0,Y 329.696,Z 449.645,A -85,B 0,C 180,E1 -15186.783,E2 -15186.783} C_VEL
LIN {X 0,Y 328.56,Z 499.887,A -85,B 0,C 180,E1 -15187.894,E2 -15187.894} C_VEL
LIN {X 0,Y 327.801,Z 513.136,A -85,B 0,C 180,E1 -15188.419,E2 -15188.419} C_VEL
LIN {X 0,Y 326.693,Z 525.316,A -85,B 0,C 180,E1 -15189.127,E2 -15189.127} C_VEL
LIN {X 0,Y 325.214,Z 537.63,A -85,B 0,C 180,E1 -15190.101,E2 -15190.101} C_VEL
LIN {X 0,Y 323.62,Z 549.307,A -85,B 0,C 180,E1 -15191.318,E2 -15191.318} C_VEL
LIN {X 0,Y 322.085,Z 559.855,A -85,B 0,C 180,E1 -15192.705,E2 -15192.705} C_VEL
LIN {X 0,Y 320.957,Z 568.532,A -85,B 0,C 180,E1 -15194.115,E2 -15194.115} C_VEL
LIN {X 0,Y 319.967,Z 576.853,A -85,B 0,C 180,E1 -15195.755,E2 -15195.755} C_VEL
LIN {X 0,Y 319.069,Z 584.46,A -85,B 0,C 180,E1 -15197.599,E2 -15197.599} C_VEL
LIN {X 0,Y 318.522,Z 591.786,A -85,B 0,C 180,E1 -15199.833,E2 -15199.833} C_VEL
LIN {X 0,Y 318.433,Z 596.708,A -85,B 0,C 180,E1 -15201.752,E2 -15201.752} C_VEL
LIN {X 0,Y 318.618,Z 600.508,A -85,B 0,C 180,E1 -15203.668,E2 -15203.668} C_VEL
LIN {X 0,Y 318.791,Z 602.479,A -85,B 0,C 180,E1 -15204.941,E2 -15204.941} C_VEL
LIN {X 0,Y 318.993,Z 603.969,A -85,B 0,C 180,E1 -15206.21,E2 -15206.21} C_VEL
LIN {X 0,Y 319.404,Z 605.703,A -85,B 0,C 180,E1 -15208.739,E2 -15208.739} C_VEL
LIN {X 0,Y 319.587,Z 605.952,A -85,B 0,C 180,E1 -15210,E2 -15210} C_VEL
LIN {X 0,Y 319.405,Z 605.697,A -85,B 0,C 180,E1 -15211.261,E2 -15211.261} C_VEL
LIN {X 0,Y 318.999,Z 603.958,A -85,B 0,C 180,E1 -15213.79,E2 -15213.79} C_VEL
LIN {X 0,Y 318.803,Z 602.463,A -85,B 0,C 180,E1 -15215.059,E2 -15215.059} C_VEL
LIN {X 0,Y 318.591,Z 599.419,A -85,B 0,C 180,E1 -15216.933,E2 -15216.933} C_VEL
LIN {X 0,Y 318.433,Z 595.17,A -85,B 0,C 180,E1 -15218.887,E2 -15218.887} C_VEL
LIN {X 0,Y 318.691,Z 588.81,A -85,B 0,C 180,E1 -15221.125,E2 -15221.125} C_VEL
LIN {X 0,Y 319.255,Z 581.918,A -85,B 0,C 180,E1 -15223.04,E2 -15223.04} C_VEL
LIN {X 0,Y 320.009,Z 575.528,A -85,B 0,C 180,E1 -15224.507,E2 -15224.507} C_VEL
LIN {X 0,Y 321.214,Z 566.615,A -85,B 0,C 180,E1 -15226.198,E2 -15226.198} C_VEL
LIN {X 0,Y 322.253,Z 558.645,A -85,B 0,C 180,E1 -15227.45,E2 -15227.45} C_VEL
LIN {X 0,Y 323.833,Z 547.853,A -85,B 0,C 180,E1 -15228.834,E2 -15228.834} C_VEL
LIN {X 0,Y 325.205,Z 537.439,A -85,B 0,C 180,E1 -15229.899,E2 -15229.899} C_VEL
LIN {X 0,Y 326.695,Z 525.031,A -85,B 0,C 180,E1 -15230.873,E2 -15230.873} C_VEL
LIN {X 0,Y 327.889,Z 511.988,A -85,B 0,C 180,E1 -15231.616,E2 -15231.616} C_VEL
LIN {X 0,Y 328.568,Z 499.302,A -85,B 0,C 180,E1 -15232.106,E2 -15232.106} C_VEL
LIN {X 0,Y 329.617,Z 447.388,A -85,B 0,C 180,E1 -15233.254,E2 -15233.254} C_VEL
LIN {X 0,Y 326.272,Z 413.893,A -85,B 0,C 180,E1 -15234.278,E2 -15234.278} C_VEL
LIN {X 0,Y 323.142,Z 388.914,A -85,B 0,C 180,E1 -15235.139,E2 -15235.139} C_VEL
LIN {X 0,Y 325.705,Z 367.677,A -85,B 0,C 180,E1 -15239.399,E2 -15239.399} C_VEL
LIN {X 0,Y 326.352,Z 361.138,A -85,B 0,C 180,E1 -15240.733,E2 -15240.733} C_VEL
LIN {X 0,Y 324.233,Z 350.55,A -85,B 0,C 180,E1 -15243.182,E2 -15243.182} C_VEL
LIN {X 0,Y 321.239,Z 338.159,A -85,B 0,C 180,E1 -15246.206,E2 -15246.206} C_VEL
LIN {X 0,Y 319.55,Z 331.786,A -85,B 0,C 180,E1 -15247.893,E2 -15247.893} C_VEL
LIN {X 0,Y 319.5,Z 331.687,A -85,B 0,C 180,E1 -15251.592,E2 -15251.592} C_VEL
LIN {X 0,Y 319.481,Z 331.652,A -85,B 0,C 180,E1 -15254.743,E2 -15254.743} C_VEL
LIN {X 0,Y 319.547,Z 331.669,A -85,B 0,C 180,E1 -15257.015,E2 -15257.015} C_VEL
LIN {X 0,Y 319.511,Z 331.662,A -85,B 0,C 180,E1 -15260.365,E2 -15260.365} C_VEL
LIN {X 0,Y 319.573,Z 331.627,A -85,B 0,C 180,E1 -15264.457,E2 -15264.457} C_VEL
LIN {X 0,Y 319.519,Z 331.686,A -85,B 0,C 180,E1 -15268.137,E2 -15268.137} C_VEL
LIN {X 0,Y 319.566,Z 331.656,A -85,B 0,C 180,E1 -15271.603,E2 -15271.603} C_VEL
LIN {X 0,Y 319.545,Z 331.681,A -85,B 0,C 180,E1 -15275.299,E2 -15275.299} C_VEL
LIN {X 0,Y 319.56,Z 331.655,A -85,B 0,C 180,E1 -15278.045,E2 -15278.045} C_VEL
LIN {X 0,Y 319.684,Z 331.647,A -85,B 0,C 180,E1 -15280.962,E2 -15280.962} C_VEL
LIN {X 0,Y 319.726,Z 331.656,A -85,B 0,C 180,E1 -15285.276,E2 -15285.276} C_VEL
LIN {X 0,Y 319.708,Z 331.655,A -85,B 0,C 180,E1 -15288.589,E2 -15288.589} C_VEL
LIN {X 0,Y 319.874,Z 331.63,A -85,B 0,C 180,E1 -15292.425,E2 -15292.425} C_VEL
LIN {X 0,Y 319.715,Z 331.648,A -85,B 0,C 180,E1 -15294.956,E2 -15294.956} C_VEL
LIN {X 0,Y 320.006,Z 331.619,A -85,B 0,C 180,E1 -15298.742,E2 -15298.742} C_VEL
LIN {X 0,Y 319.954,Z 331.624,A -85,B 0,C 180,E1 -15302.518,E2 -15302.518} C_VEL
LIN {X 0,Y 319.875,Z 331.628,A -85,B 0,C 180,E1 -15306.495,E2 -15306.495} C_VEL
LIN {X 0,Y 319.729,Z 331.656,A -85,B 0,C 180,E1 -15310.128,E2 -15310.128} C_VEL
LIN {X 0,Y 319.725,Z 331.64,A -85,B 0,C 180,E1 -15313.993,E2 -15313.993} C_VEL
LIN {X 0,Y 319.619,Z 331.671,A -85,B 0,C 180,E1 -15317.929,E2 -15317.929} C_VEL
LIN {X 0,Y 319.56,Z 331.67,A -85,B 0,C 180,E1 -15321.955,E2 -15321.955} C_VEL
LIN {X 0,Y 319.544,Z 331.67,A -85,B 0,C 180,E1 -15326.096,E2 -15326.096} C_VEL
LIN {X 0,Y 319.519,Z 331.635,A -85,B 0,C 180,E1 -15328.941,E2 -15328.941} C_VEL
LIN {X 0,Y 319.518,Z 331.658,A -85,B 0,C 180,E1 -15331.864,E2 -15331.864} C_VEL
LIN {X 0,Y 319.575,Z 331.675,A -85,B 0,C 180,E1 -15335.543,E2 -15335.543} C_VEL
LIN {X 0,Y 319.525,Z 331.647,A -85,B 0,C 180,E1 -15339.663,E2 -15339.663} C_VEL
LIN {X 0,Y 319.515,Z 331.687,A -85,B 0,C 180,E1 -15343.461,E2 -15343.461} C_VEL
LIN {X 0,Y 319.547,Z 331.653,A -85,B 0,C 180,E1 -15347.016,E2 -15347.016} C_VEL
LIN {X 0,Y 319.543,Z 331.681,A -85,B 0,C 180,E1 -15350.371,E2 -15350.371} C_VEL
LIN {X 0,Y 319.577,Z 331.675,A -85,B 0,C 180,E1 -15354.458,E2 -15354.458} C_VEL
LIN {X 0,Y 319.523,Z 331.674,A -85,B 0,C 180,E1 -15358.138,E2 -15358.138} C_VEL
LIN {X 0,Y 319.543,Z 331.645,A -85,B 0,C 180,E1 -15361.614,E2 -15361.614} C_VEL
LIN {X 0,Y 319.653,Z 331.839,A -85,B 0,C 180,E1 -15365.029,E2 -15365.029} C_VEL
LIN {X 0,Y 319.897,Z 332.911,A -85,B 0,C 180,E1 -15365.255,E2 -15365.255} C_VEL
LIN {X 0,Y 329.262,Z 353.327,A -85,B 0,C 180,E1 -15366.535,E2 -15366.535} C_VEL
LIN {X 0,Y 331.38,Z 358.274,A -85,B 0,C 180,E1 -15366.817,E2 -15366.817} C_VEL
LIN {X 0,Y 330.572,Z 413.06,A -85,B 0,C 180,E1 -15368.045,E2 -15368.045} C_VEL
LIN {X 0,Y 330.312,Z 425.972,A -85,B 0,C 180,E1 -15368.551,E2 -15368.551} C_VEL
LIN {X 0,Y 329.734,Z 439.007,A -85,B 0,C 180,E1 -15369.329,E2 -15369.329} C_VEL
LIN {X 0,Y 328.98,Z 450.226,A -85,B 0,C 180,E1 -15370.233,E2 -15370.233} C_VEL
LIN {X 0,Y 327.907,Z 460.28,A -85,B 0,C 180,E1 -15371.247,E2 -15371.247} C_VEL
LIN {X 0,Y 326.632,Z 471.122,A -85,B 0,C 180,E1 -15372.63,E2 -15372.63} C_VEL
LIN {X 0,Y 325.556,Z 479.892,A -85,B 0,C 180,E1 -15374.024,E2 -15374.024} C_VEL
LIN {X 0,Y 324.513,Z 487.918,A -85,B 0,C 180,E1 -15375.579,E2 -15375.579} C_VEL
LIN {X 0,Y 323.318,Z 495.782,A -85,B 0,C 180,E1 -15377.446,E2 -15377.446} C_VEL
LIN {X 0,Y 322.321,Z 501.693,A -85,B 0,C 180,E1 -15379.189,E2 -15379.189} C_VEL
LIN {X 0,Y 321.564,Z 507.069,A -85,B 0,C 180,E1 -15381.2,E2 -15381.2} C_VEL
LIN {X 0,Y 320.764,Z 510.962,A -85,B 0,C 180,E1 -15383.079,E2 -15383.079} C_VEL
LIN {X 0,Y 320.16,Z 513.836,A -85,B 0,C 180,E1 -15384.963,E2 -15384.963} C_VEL
LIN {X 0,Y 320.112,Z 515.178,A -85,B 0,C 180,E1 -15386.224,E2 -15386.224} C_VEL
LIN {X 0,Y 319.896,Z 516.157,A -85,B 0,C 180,E1 -15387.482,E2 -15387.482} C_VEL
LIN {X 0,Y 319.933,Z 516.737,A -85,B 0,C 180,E1 -15388.741,E2 -15388.741} C_VEL
LIN {X 0,Y 319.908,Z 516.963,A -85,B 0,C 180,E1 -15390,E2 -15390} C_VEL
LIN {X 0,Y 319.933,Z 516.777,A -85,B 0,C 180,E1 -15391.259,E2 -15391.259} C_VEL
LIN {X 0,Y 319.896,Z 516.223,A -85,B 0,C 180,E1 -15392.518,E2 -15392.518} C_VEL
LIN {X 0,Y 320.107,Z 515.271,A -85,B 0,C 180,E1 -15393.776,E2 -15393.776} C_VEL
LIN {X 0,Y 320.148,Z 513.97,A -85,B 0,C 180,E1 -15395.038,E2 -15395.038} C_VEL
LIN {X 0,Y 320.759,Z 511.145,A -85,B 0,C 180,E1 -15396.921,E2 -15396.921} C_VEL
LIN {X 0,Y 321.538,Z 507.317,A -85,B 0,C 180,E1 -15398.801,E2 -15398.801} C_VEL
LIN {X 0,Y 322.252,Z 502.237,A -85,B 0,C 180,E1 -15400.746,E2 -15400.746} C_VEL
LIN {X 0,Y 323.496,Z 494.995,A -85,B 0,C 180,E1 -15402.866,E2 -15402.866} C_VEL
LIN {X 0,Y 324.727,Z 486.966,A -85,B 0,C 180,E1 -15404.732,E2 -15404.732} C_VEL
LIN {X 0,Y 325.8,Z 478.742,A -85,B 0,C 180,E1 -15406.286,E2 -15406.286} C_VEL
LIN {X 0,Y 326.908,Z 469.705,A -85,B 0,C 180,E1 -15407.678,E2 -15407.678} C_VEL
LIN {X 0,Y 328.192,Z 459.191,A -85,B 0,C 180,E1 -15408.971,E2 -15408.971} C_VEL
LIN {X 0,Y 329.203,Z 447.672,A -85,B 0,C 180,E1 -15410.104,E2 -15410.104} C_VEL
LIN {X 0,Y 330.05,Z 436.396,A -85,B 0,C 180,E1 -15410.953,E2 -15410.953} C_VEL
LIN {X 0,Y 330.523,Z 423.908,A -85,B 0,C 180,E1 -15411.647,E2 -15411.647} C_VEL
LIN {X 0,Y 330.638,Z 413.182,A -85,B 0,C 180,E1 -15412.059,E2 -15412.059} C_VEL
LIN {X 0,Y 331.128,Z 373.741,A -85,B 0,C 180,E1 -15412.956,E2 -15412.956} C_VEL
LIN {X 0,Y 331.46,Z 358.446,A -85,B 0,C 180,E1 -15413.286,E2 -15413.286} C_VEL
LIN {X 0,Y 322.942,Z 339.341,A -85,B 0,C 180,E1 -15414.428,E2 -15414.428} C_VEL
LIN {X 0,Y 319.768,Z 332.452,A -85,B 0,C 180,E1 -15414.912,E2 -15414.912} C_VEL
LIN {X 0,Y 319.608,Z 331.722,A -85,B 0,C 180,E1 -15415.174,E2 -15415.174} C_VEL
LIN {X 0,Y 319.523,Z 331.654,A -85,B 0,C 180,E1 -15418.94,E2 -15418.94} C_VEL
LIN {X 0,Y 319.522,Z 331.674,A -85,B 0,C 180,E1 -15421.862,E2 -15421.862} C_VEL
LIN {X 0,Y 319.577,Z 331.676,A -85,B 0,C 180,E1 -15425.542,E2 -15425.542} C_VEL
LIN {X 0,Y 319.526,Z 331.683,A -85,B 0,C 180,E1 -15429.661,E2 -15429.661} C_VEL
LIN {X 0,Y 319.53,Z 331.656,A -85,B 0,C 180,E1 -15433.205,E2 -15433.205} C_VEL
LIN {X 0,Y 318.814,Z 331.751,A -85,B 0,C 180,E1 -15434.256,E2 -15434.256} C_VEL
LIN {X 0,Y 315.932,Z 332.129,A -85,B 0,C 180,E1 -15435.966,E2 -15435.966} C_VEL
LIN {X 0,Y 313.522,Z 332.431,A -85,B 0,C 180,E1 -15437.352,E2 -15437.352} C_VEL
LIN {X 0,Y 312.5,Z 332.548,A -85,B 0,C 180,E1 -15438.425,E2 -15438.425} C_VEL
LIN {X 0,Y 312.422,Z 332.551,A -85,B 0,C 180,E1 -15438.789,E2 -15438.789} C_VEL
LIN {X 0,Y 312.507,Z 332.534,A -85,B 0,C 180,E1 -15442.612,E2 -15442.612} C_VEL
LIN {X 0,Y 312.516,Z 332.554,A -85,B 0,C 180,E1 -15446.311,E2 -15446.311} C_VEL
LIN {X 0,Y 312.463,Z 332.511,A -85,B 0,C 180,E1 -15450.341,E2 -15450.341} C_VEL
LIN {X 0,Y 312.502,Z 332.548,A -85,B 0,C 180,E1 -15454.101,E2 -15454.101} C_VEL
LIN {X 0,Y 312.534,Z 332.549,A -85,B 0,C 180,E1 -15457.525,E2 -15457.525} C_VEL
LIN {X 0,Y 312.561,Z 332.549,A -85,B 0,C 180,E1 -15461.652,E2 -15461.652} C_VEL
LIN {X 0,Y 312.679,Z 332.517,A -85,B 0,C 180,E1 -15465.685,E2 -15465.685} C_VEL
LIN {X 0,Y 312.679,Z 332.534,A -85,B 0,C 180,E1 -15469.641,E2 -15469.641} C_VEL
LIN {X 0,Y 312.788,Z 332.505,A -85,B 0,C 180,E1 -15472.252,E2 -15472.252} C_VEL
LIN {X 0,Y 312.683,Z 332.536,A -85,B 0,C 180,E1 -15474.842,E2 -15474.842} C_VEL
LIN {X 0,Y 312.961,Z 332.482,A -85,B 0,C 180,E1 -15478.713,E2 -15478.713} C_VEL
LIN {X 0,Y 312.973,Z 332.494,A -85,B 0,C 180,E1 -15481.287,E2 -15481.287} C_VEL
LIN {X 0,Y 312.842,Z 332.499,A -85,B 0,C 180,E1 -15486.449,E2 -15486.449} C_VEL
LIN {X 0,Y 312.745,Z 332.526,A -85,B 0,C 180,E1 -15489.05,E2 -15489.05} C_VEL
LIN {X 0,Y 312.626,Z 332.526,A -85,B 0,C 180,E1 -15492.991,E2 -15492.991} C_VEL
LIN {X 0,Y 312.62,Z 332.542,A -85,B 0,C 180,E1 -15495.651,E2 -15495.651} C_VEL
LIN {X 0,Y 312.554,Z 332.524,A -85,B 0,C 180,E1 -15499.712,E2 -15499.712} C_VEL
LIN {X 0,Y 312.513,Z 332.545,A -85,B 0,C 180,E1 -15502.777,E2 -15502.777} C_VEL
LIN {X 0,Y 312.481,Z 332.55,A -85,B 0,C 180,E1 -15506.732,E2 -15506.732} C_VEL
LIN {X 0,Y 312.491,Z 332.546,A -85,B 0,C 180,E1 -15509.656,E2 -15509.656} C_VEL
LIN {X 0,Y 312.515,Z 332.544,A -85,B 0,C 180,E1 -15513.689,E2 -15513.689} C_VEL
LIN {X 0,Y 312.506,Z 332.558,A -85,B 0,C 180,E1 -15517.388,E2 -15517.388} C_VEL
LIN {X 0,Y 312.437,Z 332.564,A -85,B 0,C 180,E1 -15520.718,E2 -15520.718} C_VEL
LIN {X 0,Y 312.446,Z 332.53,A -85,B 0,C 180,E1 -15524.211,E2 -15524.211} C_VEL
LIN {X 0,Y 312.452,Z 332.567,A -85,B 0,C 180,E1 -15527.925,E2 -15527.925} C_VEL
LIN {X 0,Y 312.497,Z 332.741,A -85,B 0,C 180,E1 -15531.566,E2 -15531.566} C_VEL
LIN {X 0,Y 315.535,Z 344.276,A -85,B 0,C 180,E1 -15534.613,E2 -15534.613} C_VEL
LIN {X 0,Y 318.14,Z 355.677,A -85,B 0,C 180,E1 -15537.415,E2 -15537.415} C_VEL
LIN {X 0,Y 319.513,Z 362.744,A -85,B 0,C 180,E1 -15539.076,E2 -15539.076} C_VEL
LIN {X 0,Y 318.221,Z 373.376,A -85,B 0,C 180,E1 -15541.292,E2 -15541.292} C_VEL
LIN {X 0,Y 316.412,Z 387.865,A -85,B 0,C 180,E1 -15544.261,E2 -15544.261} C_VEL
LIN {X 0,Y 320.377,Z 419.783,A -85,B 0,C 180,E1 -15545.385,E2 -15545.385} C_VEL
LIN {X 0,Y 323.106,Z 448.614,A -85,B 0,C 180,E1 -15546.279,E2 -15546.279} C_VEL
LIN {X 0,Y 321.99,Z 498.912,A -85,B 0,C 180,E1 -15547.418,E2 -15547.418} C_VEL
LIN {X 0,Y 321.193,Z 512.154,A -85,B 0,C 180,E1 -15547.952,E2 -15547.952} C_VEL
LIN {X 0,Y 320.027,Z 524.328,A -85,B 0,C 180,E1 -15548.671,E2 -15548.671} C_VEL
LIN {X 0,Y 318.517,Z 536.642,A -85,B 0,C 180,E1 -15549.665,E2 -15549.665} C_VEL
LIN {X 0,Y 316.86,Z 548.317,A -85,B 0,C 180,E1 -15550.904,E2 -15550.904} C_VEL
LIN {X 0,Y 315.32,Z 558.871,A -85,B 0,C 180,E1 -15552.322,E2 -15552.322} C_VEL
LIN {X 0,Y 314.094,Z 567.541,A -85,B 0,C 180,E1 -15553.758,E2 -15553.758} C_VEL
LIN {X 0,Y 312.981,Z 575.476,A -85,B 0,C 180,E1 -15555.347,E2 -15555.347} C_VEL
LIN {X 0,Y 312.074,Z 583.464,A -85,B 0,C 180,E1 -15557.316,E2 -15557.316} C_VEL
LIN {X 0,Y 311.477,Z 590.791,A -85,B 0,C 180,E1 -15559.601,E2 -15559.601} C_VEL
LIN {X 0,Y 311.36,Z 595.714,A -85,B 0,C 180,E1 -15561.563,E2 -15561.563} C_VEL
